(* Offers algorithms used to rank features. *)
	{attribute 'TcIecLibraryType'}
{attribute 'Namespace' := 'Tc3_Vision'}
TYPE ETcVnFeatureScoreTypeORB : (
	TCVN_FST_ORB_HARRIS:=0, 	(* Harris algorithm (produces more stable keypoints, but computation takes longer). *)
	TCVN_FST_ORB_FAST:=1	(* FAST algorithm (produces slightly less stable keypoints, but computation is faster). *)
) DINT;
END_TYPE

// Data Types/Enumerations/ETcVnFlipAxis

(* Defines the axis around which to flip (mirror) the image. *)
	{attribute 'TcIecLibraryType'}
{attribute 'Namespace' := 'Tc3_Vision'}
TYPE ETcVnFlipAxis : (
	TCVN_FA_XY:=-1, 	(* Flip the image around both axes *)
	TCVN_FA_X:=0, 	(* Flip the image around the X axis *)
	TCVN_FA_Y:=1	(* Flip the image around the Y axis *)
);
END_TYPE

// Data Types/Enumerations/ETcVnFilterDirection

(* Offers directions, in which to apply filter. *)
	{attribute 'TcIecLibraryType'}
{attribute 'Namespace' := 'Tc3_Vision'}
TYPE ETcVnFilterDirection : (
	TCVN_FD_X:=0, 	(* X-direction *)
	TCVN_FD_Y:=1	(* Y-direction *)
);
END_TYPE

// Data Types/Enumerations/ETcVnFontType

(* Offers font types. *)
	{attribute 'TcIecLibraryType'}
{attribute 'Namespace' := 'Tc3_Vision'}
TYPE ETcVnFontType : (
	TCVN_FT_HERSHEY_SIMPLEX:=0, 	(* Normal size sans-serif font. *)
	TCVN_FT_HERSHEY_PLAIN:=1, 	(* Small size sans-serif font. *)
	TCVN_FT_HERSHEY_DUPLEX:=2, 	(* More complex normal size sans-serif font. *)
	TCVN_FT_HERSHEY_COMPLEX:=3, 	(* Normal size serif font. *)
	TCVN_FT_HERSHEY_TRIPLEX:=4, 	(* More complex normal size serif font. *)
	TCVN_FT_HERSHEY_COMPLEX_SMALL:=5, 	(* Small size serif font. *)
	TCVN_FT_HERSHEY_SCRIPT_SIMPLEX:=6, 	(* Hand-writing style font. *)
	TCVN_FT_HERSHEY_SCRIPT_COMPLEX:=7, 	(* More complex hand-writing style font. *)
	TCVN_FT_HERSHEY_PLAIN_ITALIC:=17, 	(* Small size sans-serif font (italic). *)
	TCVN_FT_HERSHEY_COMPLEX_ITALIC:=19, 	(* Normal size serif font (italic). *)
	TCVN_FT_HERSHEY_TRIPLEX_ITALIC:=20, 	(* More complex normal size serif font (italic). *)
	TCVN_FT_HERSHEY_COMPLEX_SMALL_ITALIC:=21	(* Small size serif font (italic). *)
) DINT;
END_TYPE

// Data Types/Enumerations/ETcVnHoughMethod

(* Offers Hough methods. *)
	{attribute 'TcIecLibraryType'}
{attribute 'Namespace' := 'Tc3_Vision'}
TYPE ETcVnHoughMethod : (
	TCVN_HM_STANDARD:=0, 	(* Classical or standard Hough transform. Every line is represented by two floating-point numbers (f1, f2), where f1 is a distance between (0,0) origin and the line, and f2 is the angle between x-axis and the normal to the line. *)
	TCVN_HM_PROBABILISTIC:=1, 	(* Probabilistic Hough transform. More efficient for pictures containing long linear segments. Returns line segments rather than the whole line, while each segment is represented by start and end point. *)
	TCVN_HM_MULTI_SCALE:=2, 	(* Multi scale variant of classical Hough transform. *)
	TCVN_HM_GRADIENT:=3, 	(* Method designed to find circles. See paper: HK Yuen, John Princen, John Illingworth, and Josef Kittler. Comparative study of hough transform methods for circle finding. Image and Vision Computing, 8(1):71–77, 1990 *)
	TCVN_HM_GRADIENT_ALT:=4	(* Variation of the GRADIENT method. *)
) DINT;
END_TYPE

// Data Types/Enumerations/ETcVnInitializableFunction

(* Offers initializable functions. *)
	{attribute 'TcIecLibraryType'}
{attribute 'Namespace' := 'Tc3_Vision'}
TYPE ETcVnInitializableFunction : (
	TCVN_IF_OCR:=0, 	(* F_VN_OCR *)
		{attribute 'hide'}
TCVN_IF_CODEDETECTION:=1	(* F_VN_CODEDETECTION *)
) DINT;
END_TYPE

// Data Types/Enumerations/ETcVnInterpolationType

(* Offers interpolation types. *)
	{attribute 'TcIecLibraryType'}
{attribute 'Namespace' := 'Tc3_Vision'}
TYPE ETcVnInterpolationType : (
	TCVN_IT_NEAREST_NEIGHBOR:=0, 	(* Nearest neighbor interpolation *)
	TCVN_IT_BILINEAR:=1, 	(* Bilinear interpolation *)
	TCVN_IT_BICUBIC:=2, 	(* Bicubic interpolation *)
	TCVN_IT_AREA_BASED:=3, 	(* Area based interpolation *)
	TCVN_IT_LANCZOS4:=4	(* Lanczos4 interpolation *)
) DINT;
END_TYPE

// Data Types/Enumerations/ETcVnKnn

(* Offers kNN model types. *)
	{attribute 'TcIecLibraryType'}
{attribute 'Namespace' := 'Tc3_Vision'}
TYPE ETcVnKnn : (
	TCVN_KNN_CLASSIFIER:=1, 	(* Classifier *)
	TCVN_KNN_NOVELTY_DETECTOR:=2, 	(* Novelty detector *)
	TCVN_KNN_REGRESSOR:=4	(* Regressor *)
) UDINT;
END_TYPE

// Data Types/Enumerations/ETcVnLineType

(* Offers line types. *)
	{attribute 'TcIecLibraryType'}
{attribute 'Namespace' := 'Tc3_Vision'}
TYPE ETcVnLineType : (
	TCVN_LT_4_CONNECTED:=4, 	(* 4-connected (pixels are connected horizontally and vertically). *)
	TCVN_LT_8_CONNECTED:=8, 	(* 8-connected (pixels are connected horizontally, vertically and diagonally). *)
	TCVN_LT_ANTIALIASED:=16	(* Antialiased (drawn using Gaussian filtering, only implemented for 8-bit images). *)
) DINT;
END_TYPE

// Data Types/Enumerations/ETcVnMorphologicalOperator

(* Offers morphological operators. *)
	{attribute 'TcIecLibraryType'}
{attribute 'Namespace' := 'Tc3_Vision'}
TYPE ETcVnMorphologicalOperator : (
	TCVN_MO_EROSION:=16#0, 	(* Shrinks objects (regions of foreground (i.e. white) pixels), removing regions smaller than the structuring element completely. *)
	TCVN_MO_DILATION:=16#1, 	(* Expands objects and thereby closes small holes inside objects. *)
	TCVN_MO_OPENING:=16#2, 	(* Applies an erosion first, a dilation second. Objects smaller than the structuring element are removed while outer shapes remain largely the same. *)
	TCVN_MO_CLOSING:=16#3, 	(* Applies a dilation first, an erosion second. Holes inside objects that fit into the structuring element are closed completely while outer shapes remain largely the same. *)
	TCVN_MO_GRADIENT:=16#4, 	(* Difference between the dilation and the erosion of an image. *)
	TCVN_MO_WHITE_TOPHAT:=16#5, 	(* Difference between an input image and its opening. *)
	TCVN_MO_BLACK_TOPHAT:=16#6, 	(* Difference between an input image and its closing. *)
	TCVN_MO_OPENING_BY_RECONSTRUCTION:=16#40000002, 	(* Opening with subsequent reconstruction of objects that were not removed by the opening. *)
	TCVN_MO_CLOSING_BY_RECONSTRUCTION:=16#40000003, 	(* Closing with subsequent reconstruction of objects that were not removed by the closing. *)
	TCVN_MO_WHITE_TOPHAT_BY_RECONSTRUCTION:=16#40000005, 	(* White tophat with subsequent reconstruction of objects that were not removed by the white tophat. *)
	TCVN_MO_BLACK_TOPHAT_BY_RECONSTRUCTION:=16#40000006	(* Black tophat with subsequent reconstruction of objects that were not removed by the black tophat. *)
) DINT;
END_TYPE

// Data Types/Enumerations/ETcVnNbc

(* Offers normal Bayes classifier types. *)
	{attribute 'TcIecLibraryType'}
{attribute 'Namespace' := 'Tc3_Vision'}
TYPE ETcVnNbc : (
	TCVN_NBC_CLASSIFIER:=1, 	(* Classifier *)
	TCVN_NBC_NOVELTY_DETECTOR:=2	(* Novelty detector *)
) UDINT;
END_TYPE

// Data Types/Enumerations/ETcVnNormalizationType

(* Offers normalization types. *)
	{attribute 'TcIecLibraryType'}
{attribute 'Namespace' := 'Tc3_Vision'}
TYPE ETcVnNormalizationType : (
	TCVN_NT_INF:=1, 	(* Infinity norm *)
	TCVN_NT_L1:=2, 	(* L1 norm *)
	TCVN_NT_L2:=4, 	(* L2 (euclidean) norm *)
	TCVN_NT_L2SQR:=5, 	(* Squared L2 norm *)
	TCVN_NT_HAMMING:=6, 	(* Hamming distance (bitwise) *)
	TCVN_NT_HAMMING2:=7, 	(* Hamming distance (each 2 bits combined to one) *)
	TCVN_NT_RELATIVE_INF:=9, 	(* Infinity norm (when comparing 2 arrays, the norm of their difference is divided by the norm of the second array) *)
	TCVN_NT_RELATIVE_L1:=10, 	(* L1 norm (when comparing 2 arrays, the norm of their difference is divided by the norm of the second array) *)
	TCVN_NT_RELATIVE_L2:=12, 	(* L2 (euclidean) norm (when comparing 2 arrays, the norm of their difference is divided by the norm of the second array) *)
	TCVN_NT_RELATIVE_L2SQR:=13, 	(* Squared L2 norm (when comparing 2 arrays, the norm of their difference is divided by the norm of the second array) *)
	TCVN_NT_RELATIVE_HAMMING:=14, 	(* Hamming distance (bitwise; when comparing 2 arrays, the norm of their difference is divided by the norm of the second array) *)
	TCVN_NT_RELATIVE_HAMMING2:=15, 	(* Hamming distance (each 2 bits combined to one; when comparing 2 arrays, the norm of their difference is divided by the norm of the second array) *)
	TCVN_NT_MINMAX:=32	(* Normalize the values to a range given by a minimum and a maximum value. *)
) DINT;
END_TYPE

// Data Types/Enumerations/ETcVnFeatureScalingType

(* Offers feature scaling  types *)
	{attribute 'TcIecLibraryType'}
{attribute 'Namespace' := 'Tc3_Vision'}
TYPE ETcVnFeatureScalingType : (
	TCVN_FST1_MAXABS:=0, 	(* Use the max of the absolute values of the feature vector. The normlized values are in the range [-1 to 1] or [0 to 1] if all the original values are positive. *)
	TCVN_FST1_MINMAX:=1, 	(* Use the min and max values of the feature vector. The normlized values are in the range [0 to 1] *)
	TCVN_FST1_STANDARDIZATION:=2	(* Use the mean and the standard deviation of the feature vector. The normalized vector has a mean value equal to zero and standard deviation equal to one *)
) DINT;
END_TYPE

// Data Types/Enumerations/ETcVnOcrModelType

(* Offers different OCR model types *)
	{attribute 'TcIecLibraryType'}
{attribute 'Namespace' := 'Tc3_Vision'}
TYPE ETcVnOcrModelType : (
	TCVN_OMT_NUMBERS:=580542139465730, 	(* Classify numbers *)
	TCVN_OMT_NUMBERS_SC:=580542139465732, 	(* Classify numbers and special characters *)
	TCVN_OMT_UCLETTERS:=580542139465736, 	(* Classify uppercase letters *)
	TCVN_OMT_NUMBERS_SC_UCLETTERS:=580542139465744	(* Classify numbers, special characters and uppercase letters *)
) ULINT;
END_TYPE

// Data Types/Enumerations/ETcVnOcrOptions

(* Provides different options to indicate whether certain actions must be performed to achieve the intended result. *)
	{attribute 'TcIecLibraryType'}
{attribute 'Namespace' := 'Tc3_Vision'}
TYPE ETcVnOcrOptions : (
	TCVN_OO_NONE:=0, 	(* No options *)
	TCVN_OO_WITHBLANKS:=1	(* Indicates that if blanks were found, they should be included in the result. By default, all blanks are omitted from the result. *)
) UDINT;
END_TYPE

// Data Types/Enumerations/ETcVnOrientationMethod

(* Offers methods to calculate the orientation of a set of points. *)
	{attribute 'TcIecLibraryType'}
{attribute 'Namespace' := 'Tc3_Vision'}
TYPE ETcVnOrientationMethod : (
	TCVN_OM_PCA:=0, 	(* Apply the PCA on the points and calculate the mean point as the center point and the rotation angle of the main principal axis *)
	TCVN_OM_FITELLIPSE:=1, 	(* Fit an ellipse around the points and calculate the center point and the rotation angle of the main axis *)
	TCVN_OM_MOMENTS:=2, 	(* Calculate the moments of the points and estimate the center and the rotation angle *)
	TCVN_OM_ENCLOSINGRECT:=3	(* Calculate a minimum area rectangle enclosing the points and calculate the center point and the rotation angle of the rectangle *)
) DINT;
END_TYPE

// Data Types/Enumerations/ETcVnPaddingMode

(* Offers padding modes. *)
	{attribute 'TcIecLibraryType'}
{attribute 'Namespace' := 'Tc3_Vision'}
TYPE ETcVnPaddingMode : (
	TCVN_PM_NONE:=0, 	(* Resize the image to the desired size without extra processing *)
	TCVN_PM_CROP_CENTER:=1, 	(* Resize and crop the image *)
	TCVN_PM_LETTERBOX:=2	(* Resize the image to the desired size while preserving the aspect ratio of the original image *)
) DINT;
END_TYPE

// Data Types/Enumerations/ETcVnPixelConnectivity

(* Offers pixel connectivities. *)
	{attribute 'TcIecLibraryType'}
{attribute 'Namespace' := 'Tc3_Vision'}
TYPE ETcVnPixelConnectivity : (
	TCVN_PC_4:=4, 	(* 4-way *)
	TCVN_PC_8:=8	(* 8-way *)
) DINT;
END_TYPE

// Data Types/Enumerations/ETcVnPrototypeClusterer

(* Offers prototype clusterer model types. *)
	{attribute 'TcIecLibraryType'}
{attribute 'Namespace' := 'Tc3_Vision'}
TYPE ETcVnPrototypeClusterer : (
	TCVN_PC_NOVELTY_DETECTOR:=2, 	(* Novelty detector *)
	TCVN_PC_CLUSTERER:=8	(* Clusterer *)
) UDINT;
END_TYPE

// Data Types/Enumerations/ETcVnRectangleIntersection

(* Offers rectangle intersection types. *)
	{attribute 'TcIecLibraryType'}
{attribute 'Namespace' := 'Tc3_Vision'}
TYPE ETcVnRectangleIntersection : (
	TCVN_RI_NONE:=0, 	(* No intersection *)
	TCVN_RI_PARTIAL:=1, 	(* Partial intersection *)
	TCVN_RI_FULL:=2	(* Full intersection *)
) DINT;
END_TYPE

// Data Types/Enumerations/ETcVnRotationAngle

(* Offers rotation angles. *)
	{attribute 'TcIecLibraryType'}
{attribute 'Namespace' := 'Tc3_Vision'}
TYPE ETcVnRotationAngle : (
	TCVN_RA_90_DEG:=0, 	(* 90 degrees *)
	TCVN_RA_180_DEG:=1, 	(* 180 degrees *)
	TCVN_RA_270_DEG:=2	(* 270 degrees *)
) DINT;
END_TYPE

// Data Types/Enumerations/ETcVnRTrees

(* Offers RTrees model types. *)
	{attribute 'TcIecLibraryType'}
{attribute 'Namespace' := 'Tc3_Vision'}
TYPE ETcVnRTrees : (
	TCVN_RT_CLASSIFIER:=1, 	(* Classifier *)
	TCVN_RT_REGRESSOR:=4	(* Regressor *)
) UDINT;
END_TYPE

// Data Types/Enumerations/ETcVnSignedNormalization

(* Offers options for normalizing images with signed data types. *)
	{attribute 'TcIecLibraryType'}
{attribute 'Namespace' := 'Tc3_Vision'}
TYPE ETcVnSignedNormalization : (
	TCVN_SN_FIX_ZERO:=0, 	(* The value 0 is fixed, i.e. the normalized image might only reach either the minimum or maximum value. *)
	TCVN_SN_FULL_SCALE:=1	(* The image is normalized to the full value range, i.e. a prior value of 0 might be != 0 after normalization. *)
);
END_TYPE

// Data Types/Enumerations/ETcVnSolvePnPMethod

(* Offers SolvePnP methods. *)
	{attribute 'TcIecLibraryType'}
{attribute 'Namespace' := 'Tc3_Vision'}
TYPE ETcVnSolvePnPMethod : (
	TCVN_SPM_ITERATIVE:=0, 	(* Levenberg-Marquardt optimization. Requires at least 4 planar or 6 non-planar reference points. *)
	TCVN_SPM_EPNP:=1, 	(* Efficient perspective-n-point camera pose estimation. Requires at least 4 reference points. *)
	TCVN_SPM_P3P:=2, 	(* Complete solution classification for the perspective-three-point problem. Requires exactly 4 reference points to find a unique solution. *)
	TCVN_SPM_AP3P:=5, 	(* An efficient algebraic solution to the perspective-three-point problem. Requires exactly 4 reference points to find a unique solution. *)
	TCVN_SPM_IPPE:=6, 	(* Infinitesimal plane-based pose estimation. Requires at least 4 coplanar reference points. *)
	TCVN_SPM_IPPE_SQUARE:=7, 	(* IPPE specialization for squares. Requires exactly 4 reference points in the following order (hsl: half square length): (-hsl, hsl, 0), (hsl, hsl, 0), (hsl, -hsl, 0), (-hsl, -hsl, 0) *)
	TCVN_SPM_SQPNP:=8	(* A consistently fast and globally optimal solution to the perspective-n-point problem. Requires at least 4 reference points. *)
) DINT;
END_TYPE

// Data Types/Enumerations/ETcVnSta

(* Offers Simplified TopoART model types. *)
	{attribute 'TcIecLibraryType'}
{attribute 'Namespace' := 'Tc3_Vision'}
TYPE ETcVnSta : (
	TCVN_STA_CLASSIFIER:=1, 	(* Classifier *)
	TCVN_STA_NOVELTY_DETECTOR:=2, 	(* Novelty detector *)
	TCVN_STA_REGRESSOR:=4, 	(* Regressor *)
	TCVN_STA_CLUSTERER:=8	(* Clusterer *)
) UDINT;
END_TYPE

// Data Types/Enumerations/ETcVnStructuringElementShape

(* Offers shapes for a structuring element. *)
	{attribute 'TcIecLibraryType'}
{attribute 'Namespace' := 'Tc3_Vision'}
TYPE ETcVnStructuringElementShape : (
	TCVN_SES_RECTANGLE:=0, 	(* Rectangle *)
	TCVN_SES_CROSS:=1, 	(* Cross *)
	TCVN_SES_ELLIPSE:=2	(* Ellipse *)
) DINT;
END_TYPE

// Data Types/Enumerations/ETcVnSvm

(* Offers SVM model types. *)
	{attribute 'TcIecLibraryType'}
{attribute 'Namespace' := 'Tc3_Vision'}
TYPE ETcVnSvm : (
	TCVN_SVM_C_CLASSIFIER:=1, 	(* Classifier *)
	TCVN_SVM_NU_CLASSIFIER:=65537, 	(* Classifier *)
	TCVN_SVM_NOVELTY_DETECTOR:=2, 	(* Novelty detector *)
	TCVN_SVM_EPS_REGRESSOR:=4, 	(* Regressor *)
	TCVN_SVM_NU_REGRESSOR:=65540	(* Regressor *)
) UDINT;
END_TYPE

// Data Types/Enumerations/ETcVnSvmKernelType

(* Offers SVM kernel types. *)
	{attribute 'TcIecLibraryType'}
{attribute 'Namespace' := 'Tc3_Vision'}
TYPE ETcVnSvmKernelType : (
	TCVN_SKT_LINEAR:=0, 	(* Linear kernel (fast) *)
	TCVN_SKT_POLY:=1, 	(* Polynomial kernel *)
	TCVN_SKT_RBF:=2, 	(* Radial basis function (RBF) kernel (good default) *)
	TCVN_SKT_SIGMOID:=3, 	(* Sigmoid kernel *)
	TCVN_SKT_CHI2:=4, 	(* Chi-squared kernel *)
	TCVN_SKT_INTER:=5	(* Histogram intersection kernel *)
) DINT;
END_TYPE

// Data Types/Enumerations/ETcVnSvmSgdClassifierType

(* Offers different types of SVMSGD classifiers. *)
	{attribute 'TcIecLibraryType'}
{attribute 'Namespace' := 'Tc3_Vision'}
TYPE ETcVnSvmSgdClassifierType : (
	TCVN_SSCT_SGD:=0, 	(* Stochastic Gradient Descent *)
	TCVN_SSCT_ASGD:=1	(* Average Stochastic Gradient Descent *)
) DINT;
END_TYPE

// Data Types/Enumerations/ETcVnSvmSgdClassifierMarginType

(* Offers different margin types for SVMSGD classifiers. *)
	{attribute 'TcIecLibraryType'}
{attribute 'Namespace' := 'Tc3_Vision'}
TYPE ETcVnSvmSgdClassifierMarginType : (
	TCVN_SSCMT_SOFT_MARGIN:=0, 	(* Soft margin allowing outliers. (beneficial for classes that cannot be separated linearly) *)
	TCVN_SSCMT_HARD_MARGIN:=1	(* Hard margin. (best-suited for linearly separable classes) *)
) DINT;
END_TYPE

// Data Types/Enumerations/ETcVnTemplateMatchMethod

(* Offers methods for template matching. *)
	{attribute 'TcIecLibraryType'}
{attribute 'Namespace' := 'Tc3_Vision'}
TYPE ETcVnTemplateMatchMethod : (
	TCVN_TMM_SQDIFF:=0, 	(* Squared difference (supports template mask) *)
	TCVN_TMM_SQDIFF_NORMED:=1, 	(* Normalized squared difference *)
	TCVN_TMM_CCORR:=2, 	(* Cross-correlation *)
	TCVN_TMM_CCORR_NORMED:=3, 	(* Normalized cross-correlation (supports template mask) *)
	TCVN_TMM_CCOEFF:=4, 	(* Correlation coefficient *)
	TCVN_TMM_CCOEFF_NORMED:=5	(* Normalized correlation coefficient *)
) DINT;
END_TYPE

// Data Types/Enumerations/ETcVnThresholdType

(* Offers threshold types. *)
	{attribute 'TcIecLibraryType'}
{attribute 'Namespace' := 'Tc3_Vision'}
TYPE ETcVnThresholdType : (
	TCVN_TT_BINARY:=0, 	(* Binary threshold *)
	TCVN_TT_BINARY_INV:=1, 	(* Inverted binary threshold *)
	TCVN_TT_TRUNC:=2, 	(* Truncated threshold (pixels > thresh are set to thresh, others keep their value) *)
	TCVN_TT_TOZERO:=3, 	(* To zero threshold (pixels < thresh are set to zero, others keep their value) *)
	TCVN_TT_TOZERO_INV:=4, 	(* Inverted to zero threshold (pixels > thresh are set to zero, others keep their value) *)
	TCVN_TT_OTSU_BINARY:=8, 	(* Binary threshold with the threshold value selected according to the Otsu algorithm *)
	TCVN_TT_OTSU_BINARY_INV:=9, 	(* Inverted binary threshold with the threshold value selected according to the Otsu algorithm *)
	TCVN_TT_OTSU_TRUNC:=10, 	(* Truncated threshold with the threshold value selected according to the Otsu algorithm *)
	TCVN_TT_OTSU_TOZERO:=11, 	(* To zero threshold with the threshold value selected according to the Otsu algorithm *)
	TCVN_TT_OTSU_TOZERO_INV:=12, 	(* Inverted to zero threshold with the threshold value selected according to the Otsu algorithm *)
	TCVN_TT_TRIANGLE_BINARY:=16, 	(* Binary threshold with the threshold value selected according to the Triangle algorithm *)
	TCVN_TT_TRIANGLE_BINARY_INV:=17, 	(* Inverted binary threshold with the threshold value selected according to the Triangle algorithm *)
	TCVN_TT_TRIANGLE_TRUNC:=18, 	(* Truncated threshold with the threshold value selected according to the Triangle algorithm *)
	TCVN_TT_TRIANGLE_TOZERO:=19, 	(* To zero threshold with the threshold value selected according to the Triangle algorithm *)
	TCVN_TT_TRIANGLE_TOZERO_INV:=20	(* Inverted to zero threshold with the threshold value selected according to the Triangle algorithm *)
) DINT;
END_TYPE

// Data Types/Enumerations/ETcVnTimestamp

(* Offers image acquisition timestamps. *)
	{attribute 'TcIecLibraryType'}
{attribute 'Namespace' := 'Tc3_Vision'}
TYPE ETcVnTimestamp : (
	TCVN_TS_IMAGE_COMPLETED:=1	(* Timestamp when the image was completed, i.e. all packets were received by the GigEVision driver. *)
) ULINT;
END_TYPE

// Data Types/Enumerations/ETcVnVectorCompareMethod

(* Offers methods for vector comparison. *)
	{attribute 'TcIecLibraryType'}
{attribute 'Namespace' := 'Tc3_Vision'}
TYPE ETcVnVectorCompareMethod : (
	TCVN_VCM_EUCLIDEAN:=0, 	(* Euclidean *)
	TCVN_VCM_ELEMENTWISE:=1	(* Elementwise *)
) DINT;
END_TYPE

// Data Types/Enumerations/ETcVnKeypointDetectionTypeAGAST

(* Offers different neighborhood types for AGAST method (For details see paper: E. Mair et al.: Adaptive and Generic Corner Detection Based on the Accelerated Segment Test, 2010). *)
	{attribute 'TcIecLibraryType'}
{attribute 'Namespace' := 'Tc3_Vision'}
TYPE ETcVnKeypointDetectionTypeAGAST : (
	TCVN_KDT_AGAST_5_8:=0, 	(* 5 of 8 *)
	TCVN_KDT_AGAST_7_12d:=1, 	(* 7 of 12 diamond *)
	TCVN_KDT_AGAST_7_12s:=2, 	(* 7 of 12 square *)
	TCVN_KDT_AGAST_9_16:=3	(* 9 of 16 *)
) DINT;
END_TYPE

// Data Types/Enumerations/ETcVnKeypointDetectionTypeFAST

(* Offers different neighborhood types for FAST method (For details see paper: E. Rosten: Machine Learning for High-speed Corner Detection, 2006). *)
	{attribute 'TcIecLibraryType'}
{attribute 'Namespace' := 'Tc3_Vision'}
TYPE ETcVnKeypointDetectionTypeFAST : (
	TCVN_KDT_FAST_5_8:=0, 	(* 5 of 8 *)
	TCVN_KDT_FAST_7_12:=1, 	(* 7 of 12 *)
	TCVN_KDT_FAST_9_16:=2	(* 9 of 16 *)
) DINT;
END_TYPE

// Data Types/Enumerations/ETcVnWorldCoordinateSystem

(* Offers world coordinate system orientations. *)
	{attribute 'TcIecLibraryType'}
{attribute 'Namespace' := 'Tc3_Vision'}
TYPE ETcVnWorldCoordinateSystem : (
	TCVN_WCS_X_RIGHT_Y_DOWN:=0, 	(* X axis points right, Y axis down (same orientation as image coordinate system) *)
	TCVN_WCS_X_DOWN_Y_RIGHT:=1, 	(* X axis points down, Y axis right *)
	TCVN_WCS_X_LEFT_Y_DOWN:=2, 	(* X axis points left, Y axis down *)
	TCVN_WCS_X_UP_Y_RIGHT:=3, 	(* X axis points up, Y axis right *)
	TCVN_WCS_X_RIGHT_Y_UP:=4, 	(* X axis points right, Y axis up *)
	TCVN_WCS_X_DOWN_Y_LEFT:=5, 	(* X axis points down, Y axis left *)
	TCVN_WCS_X_LEFT_Y_UP:=6, 	(* X axis points left, Y axis up *)
	TCVN_WCS_X_UP_Y_LEFT:=7	(* X axis points up, Y axis left *)
) DINT;
END_TYPE

// Data Types/Structs/TcVnCodeGrades1D

(* Describes code quality grades for 1D barcodes according to ISO / IEC 15416:2016. The grades range from 0 (very bad) to 4 (very good) and are averaged over several scan lines. *)
	{attribute 'TcIecLibraryType'}
{attribute 'Namespace' := 'Tc3_Vision'}
TYPE TcVnCodeGrades1D : 
	STRUCT
		(* Decode grade *)
		fDecode : REAL;
		(* Symbol contrast grade *)
		fSymbolContrast : REAL;
		(* Minimum reflectance grade *)
		fMinReflectance : REAL;
		(* Minimum edge contrast grade *)
		fMinEdgeContrast : REAL;
		(* Modulation grade *)
		fModulation : REAL;
		(* Defects grade *)
		fDefects : REAL;
		(* Decodability grade *)
		fDecodability : REAL;
		(* Overall code grade, i.e. the minimum achieved individual grade averaged over all scan lines. If different scan lines lead to different decoded data, the overall grade is 0. *)
		fOverall : REAL;
	END_STRUCT
END_TYPE

// Data Types/Structs/TcVnCodeGradesDM

(* Describes code quality grades for Data Matrix codes according to ISO / IEC 15415:2011. The grades range from 0 (very bad) to 4 (very good). *)
	{attribute 'TcIecLibraryType'}
{attribute 'Namespace' := 'Tc3_Vision'}
TYPE TcVnCodeGradesDM : 
	STRUCT
		(* Decode grade *)
		nDecode : USINT;
		(* Symbol contrast grade *)
		nSymbolContrast : USINT;
		(* Modulation grade *)
		nModulation : USINT;
		(* Reflectance margin grade *)
		nReflectanceMargin : USINT;
		(* Fixed pattern damage grade *)
		nFixedPatternDamage : USINT;
		(* Axial nonuniformity grade *)
		nAxialNonuniformity : USINT;
		(* Grid nonuniformity grade *)
		nGridNonuniformity : USINT;
		(* Unused error correction grade *)
		nUnusedErrorCorrection : USINT;
		(* Overall code grade, i.e. the minimum achieved individual grade *)
		nOverall : USINT;
	END_STRUCT
END_TYPE

// Data Types/Structs/TcVnCodeGradesQR

(* Describes code quality grades for QR codes according to ISO / IEC 15415:2011. The grades range from 0 (very bad) to 4 (very good). *)
	{attribute 'TcIecLibraryType'}
{attribute 'Namespace' := 'Tc3_Vision'}
TYPE TcVnCodeGradesQR : 
	STRUCT
		(* Decode grade *)
		nDecode : USINT;
		(* Symbol contrast grade *)
		nSymbolContrast : USINT;
		(* Modulation grade *)
		nModulation : USINT;
		(* Reflectance margin grade *)
		nReflectanceMargin : USINT;
		(* Fixed pattern damage grade *)
		nFixedPatternDamage : USINT;
		(* Axial nonuniformity grade *)
		nAxialNonuniformity : USINT;
		(* Grid nonuniformity grade *)
		nGridNonuniformity : USINT;
		(* Unused error correction grade *)
		nUnusedErrorCorrection : USINT;
		(* Format information grade *)
		nFormatInfo : USINT;
		(* Version information grade *)
		nVersionInfo : USINT;
		(* Overall code grade, i.e. the minimum achieved individual grade *)
		nOverall : USINT;
	END_STRUCT
END_TYPE

// Data Types/Structs/TcVnParamsAGAST

(* Offers parameters for AGAST method. *)
	{attribute 'TcIecLibraryType'}
{attribute 'Namespace' := 'Tc3_Vision'}
TYPE TcVnParamsAGAST : 
	STRUCT
		(* Threshold for the intensity difference between the center pixel and its surrounding circle *)
		nThreshold : DINT := 10;
		(* If true, non-maximum suppression is applied. *)
		bNonMaxSuppression : BOOL := TRUE;
		 {attribute 'hide'}
		_reserved1 : ARRAY [1..3] OF USINT;
		(* Neighborhood type *)
		 {attribute 'GUID' := 'FA6F5C56-A2E3-4BCD-8022-41680719FF8A'}
		 {attribute 'Namespace' := 'Tc3_Vision'}
		eType : ETcVnKeypointDetectionTypeAGAST := TCVN_KDT_AGAST_9_16;
	END_STRUCT
END_TYPE

// Data Types/Structs/TcVnParamsAKAZE

(* Offers parameters for AKAZE method. *)
	{attribute 'TcIecLibraryType'}
{attribute 'Namespace' := 'Tc3_Vision'}
TYPE TcVnParamsAKAZE : 
	STRUCT
		(* Type of the descriptor *)
		 {attribute 'GUID' := 'EFB57555-E4E6-46A8-8672-7CE1494D9FAA'}
		 {attribute 'Namespace' := 'Tc3_Vision'}
		eDescrType : ETcVnFeatureDescriptorTypeAKAZE := TCVN_FDT_AKAZE_MLDB;
		(* Size of the descriptor in bits (only for MLDB; 0 = full size) *)
		nDescrSize : UDINT := 0;
		(* Number of descriptor channels (currently only 3 supported for MLDB) *)
		nDescrChannels : UDINT := 3;
		(* Detector response threshold *)
		fThreshold : REAL := 0.001;
		(* Maximum octave evolution *)
		nOctaves : UDINT := 2;
		(* Number of sublevels per scale level *)
		nOctaveLayers : UDINT := 1;
		(* Diffusivity type *)
		 {attribute 'GUID' := '808733BC-B2E0-4793-A0CE-2F414F4C0F1D'}
		 {attribute 'Namespace' := 'Tc3_Vision'}
		eDiffusivity : ETcVnDiffusivityTypeKAZE := TCVN_DT1_KAZE_PM_G2;
	END_STRUCT
END_TYPE

// Data Types/Structs/TcVnParamsBlobDetection

(* Offers parameters for blob detection *)
	{attribute 'TcIecLibraryType'}
{attribute 'Namespace' := 'Tc3_Vision'}
TYPE TcVnParamsBlobDetection : 
	STRUCT
		(* Enable filtering by area (fMinArea <= area <= fMaxArea); strongly recommended to activate for filtering noise with fMinArea. *)
		bFilterByArea : BOOL := TRUE;
		(* Enable filtering by circularity (fMinCircularity <= circularity(4pi * area / perimeter^2) <= fMaxCircularity). *)
		bFilterByCircularity : BOOL := FALSE;
		(* Enable filtering by convexity (fMinConvexity <= convexity(area / hullArea) <= fMaxConvexity). *)
		bFilterByConvexity : BOOL := FALSE;
		(* Enable filtering by eccentricity (fMinEccentricity <= eccentricity <= fMaxEccentricity). *)
		bFilterByEccentricity : BOOL := FALSE;
		(* Enable filtering by inertia ratio (fMinInertiaRatio <= inertia ratio <= fMaxInertiaRatio). *)
		bFilterByInertiaRatio : BOOL := FALSE;
		 {attribute 'hide'}
		_reserved1 : ARRAY [1..3] OF USINT;
		(* Min estimated blob area in pixel *)
		fMinArea : REAL := 10;
		(* Max estimated blob area in pixel *)
		fMaxArea : REAL := 100000000;
		(* Min circularity (1.0: ideal circle, < 1: less circular, 0: not circular at all) *)
		fMinCircularity : REAL := 0;
		(* Max circularity (1.0: ideal circle, < 1: less circular, 0: not circular at all) *)
		fMaxCircularity : REAL := 1;
		(* Min convexity (1.0: blob fully convex, < 1: less convex) *)
		fMinConvexity : REAL := 0;
		(* Max convexity (1.0: blob fully convex, < 1: less convex) *)
		fMaxConvexity : REAL := 1;
		(* Min eccentricity (0.0: circular, 1.0: linear) *)
		fMinEccentricity : REAL := 0;
		(* Max eccentricity (0.0: circular, 1.0: linear) *)
		fMaxEccentricity : REAL := 1;
		(* Min inertia ratio (1.0: equal width and height, 0.0: linear) *)
		fMinInertiaRatio : REAL := 0;
		(* Max inertia ratio (1.0: equal width and height, 0.0: linear) *)
		fMaxInertiaRatio : REAL := 1;
		(* Threshold type for internally applied threshold method (OTSU_XXX only supported for USINT images). *)
		 {attribute 'GUID' := 'C40D9A7B-C720-49F8-A5B9-1663BB6925B6'}
		 {attribute 'Namespace' := 'Tc3_Vision'}
		eThresholdType : ETcVnThresholdType := TCVN_TT_BINARY;
		(* Threshold to start with (if fThresholdStep > 0, otherwise this is the only threshold used). *)
		fMinThreshold : REAL := 30;
		(* Threshold to end with (if fThresholdStep > 0, otherwise this value is not used). *)
		fMaxThreshold : REAL := 225;
		(* Sets to 0 if only 1 threshold should be used (much faster than multiple thresholds and combining the results). *)
		fThresholdStep : REAL := 0;
		(* Minimum distance between the center points of two different blobs (only used if fThresholdStep > 0; if distance < fMinBlobDistance, the blobs are treated as the same). *)
		fMinBlobDistance : REAL := 5;
		(* Minimum number of threshold steps, for which the same contour has to be detected (only used if fThresholdStep > 0; same means center point distance < fMinBlobDistance). *)
		nMinRepeatability : UDINT := 2;
		(* Selects, which of the multi-threshold blob contours should be returned. *)
		 {attribute 'GUID' := '6B3EA399-FB72-4A3D-A347-965F9D388EB6'}
		 {attribute 'Namespace' := 'Tc3_Vision'}
		eBlobCombination : ETcVnBlobCombination := TCVN_BC_MEDIAN_THRESHOLD;
	END_STRUCT
END_TYPE

// Data Types/Structs/TcVnParamsBRISK

(* Offers parameters for BRISK method. *)
	{attribute 'TcIecLibraryType'}
{attribute 'Namespace' := 'Tc3_Vision'}
TYPE TcVnParamsBRISK : 
	STRUCT
		(* Detection threshold *)
		nThreshold : DINT := 30;
		(* Detection octaves (0 for single scale) *)
		nOctaves : UDINT := 3;
		(* Scale factor for the neighborhood pattern *)
		fPatternScale : REAL := 1;
	END_STRUCT
END_TYPE

// Data Types/Structs/TcVnParamsFAST

(* Offers parameters for FAST method. *)
	{attribute 'TcIecLibraryType'}
{attribute 'Namespace' := 'Tc3_Vision'}
TYPE TcVnParamsFAST : 
	STRUCT
		(* Threshold for the intensity difference between the center pixel and its surrounding circle *)
		nThreshold : DINT := 10;
		(* If true, non-maximum suppression is applied. *)
		bNonMaxSuppression : BOOL := TRUE;
		 {attribute 'hide'}
		_reserved1 : ARRAY [1..3] OF USINT;
		(* Neighborhood type *)
		 {attribute 'GUID' := 'FBD32F44-42B6-42E8-8896-D6A6C0F64387'}
		 {attribute 'Namespace' := 'Tc3_Vision'}
		eType : ETcVnKeypointDetectionTypeFAST := TCVN_KDT_FAST_9_16;
	END_STRUCT
END_TYPE

// Data Types/Structs/TcVnParamsGFTT

(* Offers parameters for GFTT method. *)
	{attribute 'TcIecLibraryType'}
{attribute 'Namespace' := 'Tc3_Vision'}
TYPE TcVnParamsGFTT : 
	STRUCT
		(* Maximum number of corners to return (strongest ones) *)
		nMaxCorners : UDINT := 1000;
		 {attribute 'hide'}
		_reserved1 : UDINT;
		(* Minimum accepted corner quality, relative to the strongest one *)
		fQualityLevel : LREAL := 0.01;
		(* Minimum euclidean distance between returned keypoints *)
		fMinDistance : LREAL := 1;
		(* Neighborhood block size *)
		nBlockSize : UDINT := 3;
		(* If true, a Harris detector is used instead of the default method. *)
		bUseHarrisDetector : BOOL := FALSE;
		 {attribute 'hide'}
		_reserved2 : ARRAY [1..3] OF USINT;
		(* Free parameter of the Harris detector *)
		fHarrisK : LREAL := 0.04;
	END_STRUCT
END_TYPE

// Data Types/Structs/TcVnParamsKAZE

(* Offers parameters for KAZE method *)
	{attribute 'TcIecLibraryType'}
{attribute 'Namespace' := 'Tc3_Vision'}
TYPE TcVnParamsKAZE : 
	STRUCT
		(* If true, the descriptor size is extended from the default 64 byte to 128 byte. *)
		bExtended : BOOL := FALSE;
		(* If true, upright (rotation dependent) descriptors are computed. *)
		bUpright : BOOL := FALSE;
		 {attribute 'hide'}
		_reserved1 : UINT;
		(* Detector response threshold *)
		fThreshold : REAL := 0.001;
		(* Maximum octave evolution of the image *)
		nOctaves : UDINT := 4;
		(* Number of sublevels per scale level *)
		nOctaveLayers : UDINT := 2;
		(* Diffusivity type *)
		 {attribute 'GUID' := '808733BC-B2E0-4793-A0CE-2F414F4C0F1D'}
		 {attribute 'Namespace' := 'Tc3_Vision'}
		eDiffusivity : ETcVnDiffusivityTypeKAZE := TCVN_DT1_KAZE_PM_G2;
	END_STRUCT
END_TYPE

// Data Types/Structs/TcVnParamsMSER

(* Offers parameters for MSER method *)
	{attribute 'TcIecLibraryType'}
{attribute 'Namespace' := 'Tc3_Vision'}
TYPE TcVnParamsMSER : 
	STRUCT
		(* Delta for size comparison *)
		nDelta : DINT := 5;
		(* Minimum blob size *)
		nMinArea : UDINT := 60;
		(* Maximum blob size *)
		nMaxArea : UDINT := 14400;
		 {attribute 'hide'}
		_reserved1 : UDINT;
		(* Maximum blob size variation *)
		fMaxVariation : LREAL := 0.25;
		(* Minimum MSER diversity *)
		fMinDiversity : LREAL := 0.2;
		(* Maximum evolution steps (only used for color images) *)
		nMaxEvolution : UDINT := 200;
		 {attribute 'hide'}
		_reserved2 : UDINT;
		(* Area threshold to cause re-initialization (only used for color images) *)
		fAreaThreshold : LREAL := 1.01;
		(* Minimum margin (only used for color images) *)
		fMinMargin : LREAL := 0.003;
		(* Aperture size for edge bluring (only used for color images) *)
		nEdgeBlurSize : UDINT := 5;
		 {attribute 'hide'}
		_reserved3 : UDINT;
	END_STRUCT
END_TYPE

// Data Types/Structs/TcVnParamsORB

(* Offers parameters for ORB method. *)
	{attribute 'TcIecLibraryType'}
{attribute 'Namespace' := 'Tc3_Vision'}
TYPE TcVnParamsORB : 
	STRUCT
		(* Maximum number of returned keypoints *)
		nMaxPoints : UDINT := 500;
		(* Pyramid decimation ratio (must be greater than 1, should be smaller than 2) *)
		fPyramidScale : REAL := 1.2;
		(* Number of pyramid levels *)
		nPyramidLevels : UDINT := 8;
		(* Size of the border, where no features are detected (should match nPatchSize) *)
		nEdgeThreshold : UDINT := 31;
		(* First pyramid level (currently, only 0 is supported) *)
		nFirstLevel : UDINT := 0;
		(* Number of points to produce each BRIEF descriptor element (2, 3, 4) *)
		nBriefPoints : UDINT := 2;
		(* Score type (HARRIS is more stable but slightly slower than FAST) *)
		 {attribute 'GUID' := '688ACEF5-9A4A-4447-9B39-CBC4558C02DB'}
		 {attribute 'Namespace' := 'Tc3_Vision'}
		eScoreType : ETcVnFeatureScoreTypeORB := TCVN_FST_ORB_HARRIS;
		(* Patch size of the BRIEF descriptor *)
		nPatchSize : UDINT := 31;
		(* Threshold for the FAST keypoint detection *)
		nFastThreshold : DINT := 20;
	END_STRUCT
END_TYPE

// Data Types/Structs/TcVnParamsSB

(* Offers parameters for SB method (a simple blob detector with multiple thresholds). *)
	{attribute 'TcIecLibraryType'}
{attribute 'Namespace' := 'Tc3_Vision'}
TYPE TcVnParamsSB : 
	STRUCT
		(* Enable filtering by area (fMinArea <= area < fMaxArea). *)
		bFilterByArea : BOOL := TRUE;
		(* Enable filtering by circularity (fMinCircularity <= circularity(4pi * area / perimeter^2) < fMaxCircularity). *)
		bFilterByCircularity : BOOL := FALSE;
		(* Enable filtering by color (thresholdedColor(0 or 255) = nBlobColor). *)
		bFilterByColor : BOOL := FALSE;
		(* Enable filtering by convexity (fMinConvexity <= convexity(area / hullArea) < fMaxConvexity). *)
		bFilterByConvexity : BOOL := FALSE;
		(* Enable filtering by inertia ratio (fMinInertiaRatio <= inertia ratio < fMaxInertiaRatio). *)
		bFilterByInertia : BOOL := FALSE;
		 {attribute 'hide'}
		_reserved1 : ARRAY [1..3] OF USINT;
		(* Min estimated blob area in pixel *)
		fMinArea : REAL := 25;
		(* Max estimated blob area in pixel *)
		fMaxArea : REAL := 15000;
		(* Min circularity (1.0: ideal circle, < 1: less circular, 0: not circular at all) *)
		fMinCircularity : REAL := 0;
		(* Max circularity (1.0: ideal circle, < 1: less circular, 0: not circular at all) *)
		fMaxCircularity : REAL := 1;
		(* 0 or 255 *)
		nBlobColor : USINT := 255;
		 {attribute 'hide'}
		_reserved2 : ARRAY [1..3] OF USINT;
		(* Min convexity (1.0: blob fully convex, < 1: less convex) *)
		fMinConvexity : REAL := 0;
		(* Max convexity (1.0: blob fully convex, < 1: less convex) *)
		fMaxConvexity : REAL := 1;
		(* Min inertia ratio (0.0 .. 1.0) *)
		fMinInertiaRatio : REAL := 0;
		(* Max inertia ratio (0.0 .. 1.0) *)
		fMaxInertiaRatio : REAL := 1;
		(* Min distance between different blobs *)
		fMinBlobDist : REAL := 5;
		(* Min number of same detected blobs (dist < fMinBlobDist) in different thresholds *)
		nMinRepeatability : UDINT := 2;
		(* Min threshold (start) *)
		fMinThreshold : REAL := 30;
		(* Max threshold (stop) *)
		fMaxThreshold : REAL := 225;
		(* Threshold step between min and max threshold *)
		fThresholdStep : REAL := 10;
	END_STRUCT
END_TYPE

// Version/Global_Version
{attribute 'TcGenerated'}
// This function has been automatically generated from the project information.
VAR_GLOBAL CONSTANT
	{attribute 'const_non_replaced'}
	{attribute 'linkalways'}
	stLibVersion_Tc3_Vision : ST_LibVersion := (iMajor := 5, iMinor := 5, iBuild := 10, iRevision := 0, sVersion := '5.5.10.0');
	{attribute 'const_non_replaced'}
	{attribute 'linkalways'}
	sLibraryId_Tc3_Vision : String := 'Beckhoff Automation GmbH|Tc3_Vision|5.5.10.0';
END_VAR

// Global Variables/Global_Variables

	VAR_GLOBAL
		VISION_ADS_TIMEOUT	:	TIME := TIME#5s;	(* Default ADS timeout. *)
	END_VAR

// Global Variables/TC3_VISION_IID_LIST

	VAR_GLOBAL
		IID_ITcVnColorModel	:	IID := (Data1 := 16#AFF801F3, Data2 := 16#60D0, Data3 := 16#43FA, Data4 := [16#98, 16#0F, 16#57, 16#2A, 16#62, 16#05, 16#B5, 16#AF]);	(* Interface ID for interface ITcVnColorModel *)
	END_VAR

// Function Blocks/Image Acquisition/FB_VN_GevCameraControl

	{attribute 'c++_compatible'}
	{attribute 'external_name' := 'FB_VN_GevCameraControl_GUID_E0C38C9A_95D7_4F88_D282_FD5E0D0B8646'}
	{attribute 'TcIecLibraryType'}
	{attribute 'no_explicit_call' :='do not call this POU directly'}
	(* This FB provides the basic functionality to control a GigE Vision camera and access its calibration data. *)
	FUNCTION_BLOCK FB_VN_GevCameraControl
	VAR
		(* Internal reference to the corresponding TcVnGevImageProvider TcCOM module ID, which needs to be set via TC init symbol. *)
		{attribute 'TcInitSymbol'}
		{attribute 'TcCategoryOID' := 'TcVnGevImageProvider'}
		 {attribute 'GUID' := '18071995-0000-0000-0000-00000000000F'}
		oidITcVnGevImageProvider : OTCID;
		 {attribute 'hide'}
		_reserved1 : UINT_0_32;
		(* Internal stuff *)
		{attribute 'hide'}
		 {attribute 'GUID' := '18071995-0000-0000-0000-000000000018'}
		pInternal : PVOID;
	END_VAR


	(* Delete all images contained in the TcVnGevImageProvider TcCOM module receive queue and reset the corresponding omitted images counter. *)
	METHOD ClearImageQueue : HRESULT
END_METHOD


	(* Close the control channel to the camera. *)
	METHOD CloseCamera : HRESULT
END_METHOD


	(* Internal method *)
	{attribute 'hide'}
	METHOD FB_exit : BOOL
	VAR_INPUT
		(*  if TRUE, the exit method is called for exiting an instance that is copied afterwards (online change). *)
		bInCopyCode : BOOL;
	END_VAR
END_METHOD


	(* Internal method *)
	{attribute 'hide'}
	METHOD FB_init : BOOL
	VAR_INPUT
		(*  if TRUE, the retain variables are initialized (warm start / cold start) *)
		bInitRetains : BOOL;
		(*  if TRUE, the instance afterwards gets moved into the copy code (online change) *)
		bInCopyCode : BOOL;
	END_VAR
END_METHOD


	(* Gets the reference calibration pattern points from the TcVnGevImageProvider TcCOM module (Can be set from the calibration assistant) *)
	METHOD GetCalibPatternRef : HRESULT
	VAR_INPUT
		(* Returns the reference calibration pattern points (ContainerType_Vector_TcVnPoint3_REAL) *)
 {attribute 'GUID' := 'BC72B333-E095-465B-9693-7979773CA3B8'}
				ipCalibPatternRef : REFERENCE TO ITcVnContainer;
	END_VAR
END_METHOD


	(* Gets the camera matrix from the TcVnGevImageProvider TcCOM module (requires intrinsic calibration parameters, e.g. set by the calibration assistant) *)
	METHOD GetCameraMatrix : HRESULT
	VAR_IN_OUT
		(* Returns the camera matrix *)
 {attribute 'GUID' := '91A420A3-4727-4481-B3BB-170528E5BC7C'}
		 {attribute 'Namespace' := 'VN'}
				aCameraMatrix : TcVnMatrix3x3_LREAL;
	END_VAR
END_METHOD


	(* Gets the current available image (first in receive queue). *)
	METHOD GetCurrentImage : HRESULT
	VAR_INPUT
		(* Returns the image *)
 {attribute 'GUID' := '70D42C6D-6F4E-4719-8B29-2883D5D59B1C'}
				ipImage : REFERENCE TO ITcVnImage;
	END_VAR
END_METHOD


	(* Gets the current available image (first in receive queue) with undistortion applied. Incompatible with pixel formats that contain an encoding, e.g. a Bayer pattern. Requires intrinsic calibration parameters in the TcVnGevImageProvider TcCOM module, e.g. set by the calibration assistant. *)
	METHOD GetCurrentImageUndistorted : HRESULT
	VAR_INPUT
		(* Returns the undistorted image *)
 {attribute 'GUID' := '70D42C6D-6F4E-4719-8B29-2883D5D59B1C'}
				ipImage : REFERENCE TO ITcVnImage;
	END_VAR
END_METHOD


	(* Gets the current available image (first in receive queue) and its corresponding GVSP info. *)
	METHOD GetCurrentImageWithGvspInfo : HRESULT
	VAR_INPUT
		(* Returns the image *)
 {attribute 'GUID' := '70D42C6D-6F4E-4719-8B29-2883D5D59B1C'}
				ipImage : REFERENCE TO ITcVnImage;
	END_VAR
	VAR_IN_OUT
		(* Returns the GVSP info *)
 {attribute 'GUID' := '63FC7E33-91CD-44CD-9015-0BD1DC25722C'}
				stGvspInfo : GVSP_IMAGE_INFO;
	END_VAR
END_METHOD


	(* Gets the current available image (first in receive queue) with its corresponding GVSP info and undistortion applied. Incompatible with pixel formats that contain an encoding, e.g. a Bayer pattern. Requires intrinsic calibration parameters in the TcVnGevImageProvider TcCOM module, e.g. set by the calibration assistant. *)
	METHOD GetCurrentImageWithGvspInfoUndistorted : HRESULT
	VAR_INPUT
		(* Returns the undistorted image *)
 {attribute 'GUID' := '70D42C6D-6F4E-4719-8B29-2883D5D59B1C'}
				ipImage : REFERENCE TO ITcVnImage;
	END_VAR
	VAR_IN_OUT
		(* Returns the GVSP info *)
 {attribute 'GUID' := '63FC7E33-91CD-44CD-9015-0BD1DC25722C'}
				stGvspInfo : GVSP_IMAGE_INFO;
	END_VAR
END_METHOD


	(* Gets the current available image (first in receive queue) and corresponding timestamps. *)
	METHOD GetCurrentImageWithTimestamps : HRESULT
	VAR_INPUT
		(* Returns the image *)
 {attribute 'GUID' := '70D42C6D-6F4E-4719-8B29-2883D5D59B1C'}
				ipImage : REFERENCE TO ITcVnImage;
		(* Select timestamps to return (ETcVnTimestamp) *)
		nTimestamps : ULINT;
		(* Returns the requested timestamps (make sure to provide an array of sufficient size). *)
		pTimestamps : POINTER TO LINT;
	END_VAR
	VAR_OUTPUT
		(* Returns the GVSP info *)
 {attribute 'GUID' := '63FC7E33-91CD-44CD-9015-0BD1DC25722C'}
				stGvspInfo : GVSP_IMAGE_INFO;
	END_VAR
END_METHOD


	(* Gets the distortion coefficients from the TcVnGevImageProvider TcCOM module (requires intrinsic calibration parameters, e.g. set by the calibration assistant) *)
	METHOD GetDistortionCoefficients : HRESULT
	VAR_IN_OUT
		(* Returns the distortion coefficients [k1, k2, p1, p2, k3, k4, k5, k6] *)
 {attribute 'GUID' := 'DD112102-C23A-4B37-A43A-A96400B57010'}
		 {attribute 'Namespace' := 'VN'}
				aDistortionCoefficients : TcVnArray8_LREAL;
	END_VAR
END_METHOD


	(* Gets the last received image from the queue. *)
	METHOD GetLastImageFromQueue : HRESULT
	VAR_INPUT
		(* Returns the image *)
 {attribute 'GUID' := '70D42C6D-6F4E-4719-8B29-2883D5D59B1C'}
				ipImage : REFERENCE TO ITcVnImage;
	END_VAR
END_METHOD


	(* Gets the number of omitted images since the last call of ClearImageQueue(). If the image receive queue in the TcVnGevImageProvider TcCOM module is full and a new image arrives, the first one in the queue will be deleted and the omitted counter is increased. *)
	METHOD GetOmittedImagesNum : HRESULT
	VAR_IN_OUT
		(* Returns the number of omitted images *)
		nOmitted : ULINT;
	END_VAR
END_METHOD


	(* Gets the rotation matrix from the TcVnGevImageProvider TcCOM module (requires extrinsic calibration parameters, e.g. set by the calibration assistant) *)
	METHOD GetRotationMatrix : HRESULT
	VAR_IN_OUT
		(* Returns the rotation matrix *)
 {attribute 'GUID' := '91A420A3-4727-4481-B3BB-170528E5BC7C'}
		 {attribute 'Namespace' := 'VN'}
				aRotationMatrix : TcVnMatrix3x3_LREAL;
	END_VAR
END_METHOD


	(* Gets the current state of the internal camera control state machine. *)
	METHOD GetState : ETcVnCameraState
END_METHOD


	(* Gets the translation vector from the TcVnGevImageProvider TcCOM module (requires extrinsic calibration parameters, e.g. set by the calibration assistant) *)
	METHOD GetTranslationVector : HRESULT
	VAR_IN_OUT
		(* Returns the translation vector *)
 {attribute 'GUID' := 'B9A67DEB-A7D1-4F25-95A3-4A82FA5C1E28'}
		 {attribute 'Namespace' := 'VN'}
				aTranslationVector : TcVnVector3_LREAL;
	END_VAR
END_METHOD


	(* Initialize the camera to the intended state (includes sending the 'InitCameraCommands' defined in the GevImageAcquisition TcCOM module to the camera). *)
	METHOD InitializeCamera : HRESULT
END_METHOD


	(* Open a control channel to the camera. *)
	METHOD OpenCamera : HRESULT
END_METHOD


	(* Reset the camera controller to initial state (might require multiple calls depending on current state, until S_OK is returned) *)
	METHOD Reset : HRESULT
END_METHOD


	(* Reset the camera features to initial state (sends the 'InitCameraCommands' defined in the GevImageAcquisition TcCOM module to the camera). *)
	METHOD ResetCameraFeatures : HRESULT
END_METHOD


	(* Sets the camera matrix to the TcVnGevImageProvider TcCOM module *)
	METHOD SetCameraMatrix : HRESULT
	VAR_IN_OUT
		(* The camera matrix to be copied to the TcCOM module *)
 {attribute 'GUID' := '91A420A3-4727-4481-B3BB-170528E5BC7C'}
		 {attribute 'Namespace' := 'VN'}
				aCameraMatrix : TcVnMatrix3x3_LREAL;
	END_VAR
END_METHOD


	(* Sets the distortion coefficients to the TcVnGevImageProvider TcCOM module *)
	METHOD SetDistortionCoefficients : HRESULT
	VAR_IN_OUT
		(* The distortion coefficients to be copied to the TcCOM module *)
 {attribute 'GUID' := 'DD112102-C23A-4B37-A43A-A96400B57010'}
		 {attribute 'Namespace' := 'VN'}
				aDistortionCoefficients : TcVnArray8_LREAL;
	END_VAR
END_METHOD


	(* Sets the rotation matrix to the TcVnGevImageProvider TcCOM module *)
	METHOD SetRotationMatrix : HRESULT
	VAR_IN_OUT
		(* The rotation matrix to be copied to the TcCOM module *)
 {attribute 'GUID' := '91A420A3-4727-4481-B3BB-170528E5BC7C'}
		 {attribute 'Namespace' := 'VN'}
				aRotationMatrix : TcVnMatrix3x3_LREAL;
	END_VAR
END_METHOD


	(* Sets the translation vector to the TcVnGevImageProvider TcCOM module *)
	METHOD SetTranslationVector : HRESULT
	VAR_IN_OUT
		(* The translation vector to be copied to the TcCOM module *)
 {attribute 'GUID' := 'B9A67DEB-A7D1-4F25-95A3-4A82FA5C1E28'}
		 {attribute 'Namespace' := 'VN'}
				aTranslationVector : TcVnVector3_LREAL;
	END_VAR
END_METHOD


	(* Send the 'StartAcquisitionCommands' defined in the TcVnGevImageProvider TcCOM module to the camera. *)
	METHOD StartAcquisition : HRESULT
END_METHOD


	(* Send the 'StopAcquisitionCommands' defined in the TcVnGevImageProvider TcCOM module to the camera. *)
	METHOD StopAcquisition : HRESULT
END_METHOD


	(* Send the 'SoftwareTriggerCommands' defined in the TcVnGevImageProvider TcCOM module to the camera. *)
	METHOD TriggerImage : HRESULT
END_METHOD

END_FUNCTION_BLOCK

// Function Blocks/Image Acquisition/FB_VN_FileSourceControl

	{attribute 'c++_compatible'}
	{attribute 'external_name' := 'FB_VN_FileSourceControl_GUID_BF1EF806_AD3C_426D_E484_B59DB5FAA980'}
	{attribute 'TcIecLibraryType'}
	{attribute 'no_explicit_call' :='do not call this POU directly'}
	(* This FB provides access to the images send by a File Source instance. *)
	FUNCTION_BLOCK FB_VN_FileSourceControl
	VAR
		(* Internal reference to the corresponding TcVnFileImageProvider TcCOM module ID, which needs to be set via TC init symbol. *)
		{attribute 'TcInitSymbol'}
		{attribute 'TcCategoryOID' := 'TcVnFileImageProvider'}
		 {attribute 'GUID' := '18071995-0000-0000-0000-00000000000F'}
		oidITcVnFileImageProvider : OTCID;
		 {attribute 'hide'}
		_reserved1 : UINT_0_32;
		(* Internal reference to private data. *)
		{attribute 'hide'}
		 {attribute 'GUID' := '18071995-0000-0000-0000-000000000018'}
		pPriv : PVOID;
	END_VAR


	(* Internal method *)
	{attribute 'hide'}
	METHOD FB_exit : BOOL
	VAR_INPUT
		(* If TRUE, the exit method is called for exiting an instance that is copied afterwards (online change). *)
		bInCopyCode : BOOL;
	END_VAR
END_METHOD


	(* Internal method *)
	{attribute 'hide'}
	METHOD FB_init : BOOL
	VAR_INPUT
		(* If TRUE, the retain variables are initialized (warm start / cold start) *)
		bInitRetains : BOOL;
		(* If TRUE, the exit method is called for exiting an instance that is copied afterwards (online change). *)
		bInCopyCode : BOOL;
	END_VAR
END_METHOD


	(* Gets the current available image (if any). *)
	METHOD GetCurrentImage : HRESULT
	VAR_INPUT
		(* Returns the image *)
 {attribute 'GUID' := '70D42C6D-6F4E-4719-8B29-2883D5D59B1C'}
				ipImage : REFERENCE TO ITcVnImage;
	END_VAR
END_METHOD


	(* Gets the current available image (if any) and the corresponding file name. *)
	METHOD GetCurrentImageAndFileName : HRESULT
	VAR_INPUT
		(* Returns the image *)
 {attribute 'GUID' := '70D42C6D-6F4E-4719-8B29-2883D5D59B1C'}
				ipImage : REFERENCE TO ITcVnImage;
	END_VAR
	VAR_IN_OUT CONSTANT
		(* Returns the file name *)
 {attribute 'GUID' := '18071995-0000-0000-0000-00000000001A'}
				sFileName : STRING;
	END_VAR
	VAR_INPUT
		(* Define the maximum allowed length for the file name *)
		nMaxLen : UINT;
	END_VAR
END_METHOD


	(* Activates the File Source. If not in trigger mode, it will start sending images. *)
	METHOD StartAcquisition : HRESULT
END_METHOD


	(* Deactivates the File Source. It will stop sending images. *)
	METHOD StopAcquisition : HRESULT
END_METHOD


	(* Reset the controller to initial state (might require multiple calls depending on current state, until S_OK is returned) *)
	METHOD Reset : HRESULT
END_METHOD


	(* Gets the current state of the internal camera control state machine. *)
	METHOD GetState : ETcVnCameraState
END_METHOD


	(* If in trigger mode, this function triggers the next image in the list. *)
	METHOD TriggerImage : HRESULT
END_METHOD


	(* If in trigger mode, this function triggers a specific image in the list. *)
	METHOD TriggerImageExp : HRESULT
	VAR_INPUT
		(* Amount of images to skip, relative to current *)
		nSkipImages : DINT;
	END_VAR
END_METHOD


	(* If in trigger mode, this function triggers a specific image in the list by name. *)
	METHOD TriggerImageByName : HRESULT
	VAR_IN_OUT CONSTANT
		(* Name of the image to trigger *)
 {attribute 'GUID' := '18071995-0000-0000-0000-00000000001A'}
				sImageName : STRING;
	END_VAR
END_METHOD

END_FUNCTION_BLOCK

// Function Blocks/Image Acquisition/FB_VN_SimpleCameraControl

	{attribute 'c++_compatible'}
	{attribute 'external_name' := 'FB_VN_SimpleCameraControl_GUID_3530661D_FCB1_48FD_F78A_F761ECBA890C'}
	{attribute 'TcIecLibraryType'}
	{attribute 'no_explicit_call' :='do not call this POU directly'}
	(* This FB provides the basic functionality to control a camera or a FileSource. *)
	FUNCTION_BLOCK FB_VN_SimpleCameraControl
	VAR
		(* Internal reference to the corresponding TcVnImageProvider TcCOM module ID, which needs to be set via TC init symbol. *)
		{attribute 'TcInitSymbol'}
		{attribute 'TcCategoryOID' := 'TcVnImageProvider'}
		 {attribute 'GUID' := '18071995-0000-0000-0000-00000000000F'}
		oidITcVnImageProvider : OTCID;
		 {attribute 'hide'}
		_reserved1 : UINT_0_32;
		(* Internal stuff *)
		{attribute 'hide'}
		 {attribute 'GUID' := '18071995-0000-0000-0000-000000000018'}
		pInternal : PVOID;
	END_VAR


	(* Internal method *)
	{attribute 'hide'}
	METHOD FB_exit : BOOL
	VAR_INPUT
		(*  if TRUE, the exit method is called for exiting an instance that is copied afterwards (online change). *)
		bInCopyCode : BOOL;
	END_VAR
END_METHOD


	(* Internal method *)
	{attribute 'hide'}
	METHOD FB_init : BOOL
	VAR_INPUT
		(*  if TRUE, the retain variables are initialized (warm start / cold start) *)
		bInitRetains : BOOL;
		(*  if TRUE, the instance afterwards gets moved into the copy code (online change) *)
		bInCopyCode : BOOL;
	END_VAR
END_METHOD


	(* Get the current available image (if any). *)
	METHOD GetCurrentImage : HRESULT
	VAR_INPUT
		(* Returns the image *)
 {attribute 'GUID' := '70D42C6D-6F4E-4719-8B29-2883D5D59B1C'}
				ipImage : REFERENCE TO ITcVnImage;
	END_VAR
END_METHOD


	(* Get the current state of the internal camera control state machine. *)
	METHOD GetState : ETcVnCameraState
END_METHOD


	(* Reset the camera to initial state (might require multiple calls depending on current state, until S_OK is returned) *)
	METHOD Reset : HRESULT
END_METHOD


	(* Start the image acquisition. *)
	METHOD StartAcquisition : HRESULT
END_METHOD


	(* Stop the image acquisition. *)
	METHOD StopAcquisition : HRESULT
END_METHOD


	(* Trigger the next image. *)
	METHOD TriggerImage : HRESULT
END_METHOD

END_FUNCTION_BLOCK

// Function Blocks/File Access/FB_VN_InitializeFunction

	{attribute 'c++_compatible'}
	{attribute 'external_name' := 'FB_VN_InitializeFunction_GUID_C13A97AB_8F2F_4225_FF15_35BCADA0C9FC'}
	{attribute 'TcIecLibraryType'}
	(* This FB initializes selected functions. Before, it needs to initialize itself, i.e. call the FB until the output bInitialized is true before using it for function initialization. *)
	FUNCTION_BLOCK FB_VN_InitializeFunction
	VAR_INPUT
		(* Selects the function to initialize *)
		 {attribute 'GUID' := 'E6ED44CE-C5A2-4A6C-A74A-99081CD9253B'}
		 {attribute 'Namespace' := 'Tc3_Vision'}
		eFunction : ETcVnInitializableFunction;
	END_VAR
	VAR
		 {attribute 'hide'}
		_reserved1 : UINT_0_32;
	END_VAR
	VAR_INPUT
		(* Selects initialization options for the function *)
		nOptions : ULINT := 0;
		(* Function initialization is triggered by a rising edge at this input. *)
		bStart : BOOL;
	END_VAR
	VAR
		 {attribute 'hide'}
		_reserved2 : ARRAY [1..3] OF USINT;
	END_VAR
	VAR_INPUT
		(* Indicates the time before the function is cancelled. *)
		nTimeout : TIME := VISION_ADS_TIMEOUT;
	END_VAR
	VAR_OUTPUT
		(* This output remains TRUE until the function block has executed a command, but at the longest for the duration supplied to the 'nTimeout' input. While bBusy = TRUE, no new command will be accepted at the inputs. *)
		bBusy : BOOL;
		(* This output is switched to TRUE as soon as an error occurs during the execution of a command. The command-specific error code is contained in ‘nErrorId’. If the function block has a timeout error, 'bError' is TRUE and 'nErrorId' is 1861 (hexadecimal 0x745). Is reset to FALSE by the execution of a command at the inputs. *)
		bError : BOOL;
	END_VAR
	VAR
		 {attribute 'hide'}
		_reserved3 : UINT;
	END_VAR
	VAR_OUTPUT
		(* Contains the ADS error code or the command-specific error code of the last executed command. Is reset to 0 by the execution of a command at the inputs. *)
		nErrorId : UDINT;
	END_VAR
	VAR
		(* Internal parameter *)
		{attribute 'hide'}
		nAdsInvStamp : UINT;
		(* Internal parameter *)
		{attribute 'hide'}
		nAdsInvCnt : BYTE;
		(* Internal parameter *)
		{attribute 'hide'}
		ePendingRequest : BYTE;
		(* Internal parameter *)
		{attribute 'hide'}
		nTimeElapsed : TIME;
		(* Internal parameter *)
		{attribute 'hide'}
		bLastRead : BOOL;
		 {attribute 'hide'}
		_reserved4 : UINT_24_56;
		(* Internal parameter *)
		{attribute 'hide'}
		 {attribute 'GUID' := '18071995-0000-0000-0000-000000000018'}
		pBuffer : PVOID;
		(* Internal parameter *)
		{attribute 'hide'}
		 {attribute 'GUID' := 'E6ED44CE-C5A2-4A6C-A74A-99081CD9253B'}
		 {attribute 'Namespace' := 'Tc3_Vision'}
		ePendingFunction : ETcVnInitializableFunction;
		 {attribute 'hide'}
		_reserved5 : UDINT;
		(* Internal parameter *)
		{attribute 'hide'}
		nPendingOptions : ULINT;
		(* Internal parameter *)
		{attribute 'hide'}
		 {attribute 'GUID' := '18071995-0000-0000-0000-000000000018'}
		pFilePathPending : PVOID;
		(* Internal parameter *)
		{attribute 'hide'}
		nFilePathCounter : DINT;
		 {attribute 'hide'}
		_reserved6 : UINT_0_32;
	END_VAR


	(* Internal method *)
	{attribute 'hide'}
	METHOD FB_exit : BOOL
	VAR_INPUT
		(*  if TRUE, the exit method is called for exiting an instance that is copied afterwards (online change). *)
		bInCopyCode : BOOL;
	END_VAR
END_METHOD


	(* Internal method *)
	{attribute 'hide'}
	METHOD FB_init : BOOL
	VAR_INPUT
		(*  if TRUE, the retain variables are initialized (warm start / cold start) *)
		bInitRetains : BOOL;
		(*  if TRUE, the instance afterwards gets moved into the copy code (online change) *)
		bInCopyCode : BOOL;
	END_VAR
END_METHOD

END_FUNCTION_BLOCK

// Function Blocks/File Access/FB_VN_ReadCalibrationPattern

	{attribute 'c++_compatible'}
	{attribute 'external_name' := 'FB_VN_ReadCalibrationPattern_GUID_0334E03E_2BBE_407D_E2A1_068B13B2E811'}
	{attribute 'TcIecLibraryType'}
	(* This FB reads calibration pattern reference points from an xml file on the targte pc. *)
	FUNCTION_BLOCK FB_VN_ReadCalibrationPattern
	VAR_IN_OUT CONSTANT
		(* Full path of the file or relative path to the default directory on the target pc *)
		 {attribute 'GUID' := '18071995-0000-0000-0000-00000000001A'}
		sFilePath : STRING;
	END_VAR
	VAR_INPUT
		(* Returns a container with the pattern points (ContainerType_Vector_TcVnPoint3_REAL) *)
		 {attribute 'GUID' := 'BC72B333-E095-465B-9693-7979773CA3B8'}
		ipDestContainer : REFERENCE TO ITcVnContainer;
		(* Reading the file is triggered by a rising edge at this input. *)
		bRead : BOOL;
	END_VAR
	VAR
		 {attribute 'hide'}
		_reserved1 : ARRAY [1..3] OF USINT;
	END_VAR
	VAR_INPUT
		(* Indicates the time before the function is cancelled. *)
		nTimeout : TIME := VISION_ADS_TIMEOUT;
	END_VAR
	VAR_OUTPUT
		(* This output remains TRUE until the function block has executed a command, but at the longest for the duration supplied to the 'nTimeout' input. While bBusy = TRUE, no new command will be accepted at the inputs. *)
		bBusy : BOOL;
		(* This output is switched to TRUE as soon as an error occurs during the execution of a command. The command-specific error code is contained in ‘nErrorId’. If the function block has a timeout error, 'bError' is TRUE and 'nErrorId' is 1861 (hexadecimal 0x745). Is reset to FALSE by the execution of a command at the inputs. *)
		bError : BOOL;
	END_VAR
	VAR
		 {attribute 'hide'}
		_reserved2 : UINT;
	END_VAR
	VAR_OUTPUT
		(* Contains the ADS error code or the command-specific error code of the last executed command. Is reset to 0 by the execution of a command at the inputs. *)
		nErrorId : UDINT;
	END_VAR
	VAR
		(* Internal parameter *)
		{attribute 'hide'}
		nAdsInvStamp : UINT;
		(* Internal parameter *)
		{attribute 'hide'}
		nAdsInvCnt : BYTE;
		(* Internal parameter *)
		{attribute 'hide'}
		ePendingRequest : BYTE;
		(* Internal parameter *)
		{attribute 'hide'}
		nTimeElapsed : TIME;
		(* Internal parameter *)
		{attribute 'hide'}
		bLastRead : BOOL;
		 {attribute 'hide'}
		_reserved3 : UINT_24_56;
		(* Internal parameter *)
		{attribute 'hide'}
		 {attribute 'GUID' := '18071995-0000-0000-0000-000000000018'}
		pBuffer : PVOID;
		(* Internal parameter *)
		{attribute 'hide'}
		 {attribute 'GUID' := '18071995-0000-0000-0000-000000000018'}
		pFilePathPending : PVOID;
	END_VAR


	(* Internal method *)
	{attribute 'hide'}
	METHOD FB_exit : BOOL
	VAR_INPUT
		(*  if TRUE, the exit method is called for exiting an instance that is copied afterwards (online change). *)
		bInCopyCode : BOOL;
	END_VAR
END_METHOD


	(* Internal method *)
	{attribute 'hide'}
	METHOD FB_init : BOOL
	VAR_INPUT
		(*  if TRUE, the retain variables are initialized (warm start / cold start) *)
		bInitRetains : BOOL;
		(*  if TRUE, the instance afterwards gets moved into the copy code (online change) *)
		bInCopyCode : BOOL;
	END_VAR
END_METHOD

END_FUNCTION_BLOCK

// Function Blocks/File Access/FB_VN_ReadCalibrationResult

	{attribute 'c++_compatible'}
	{attribute 'external_name' := 'FB_VN_ReadCalibrationResult_GUID_EE7898B1_588B_4444_D687_3E4CD4FF96B9'}
	{attribute 'TcIecLibraryType'}
	(* This FB reads calibration results from a json file on the targte pc. *)
	FUNCTION_BLOCK FB_VN_ReadCalibrationResult
	VAR_IN_OUT CONSTANT
		(* Full path of the file or relative path to the default directory on the target pc *)
		 {attribute 'GUID' := '18071995-0000-0000-0000-00000000001A'}
		sFilePath : STRING;
	END_VAR
	VAR_INPUT
		(* Returns the camera matrix *)
		 {attribute 'GUID' := '91A420A3-4727-4481-B3BB-170528E5BC7C'}
		 {attribute 'Namespace' := 'VN'}
		aCameraMatrix : REFERENCE TO TcVnMatrix3x3_LREAL;
		(* Returns the distortion coefficients *)
		 {attribute 'GUID' := 'DD112102-C23A-4B37-A43A-A96400B57010'}
		 {attribute 'Namespace' := 'VN'}
		aDistortionCoefficients : REFERENCE TO TcVnArray8_LREAL;
		(* Returns the rotation matrix *)
		 {attribute 'GUID' := '91A420A3-4727-4481-B3BB-170528E5BC7C'}
		 {attribute 'Namespace' := 'VN'}
		aRotationMatrix : REFERENCE TO TcVnMatrix3x3_LREAL;
		(* Returns the translation vector *)
		 {attribute 'GUID' := 'B9A67DEB-A7D1-4F25-95A3-4A82FA5C1E28'}
		 {attribute 'Namespace' := 'VN'}
		aTranslationVector : REFERENCE TO TcVnVector3_LREAL;
		(* Reading the file is triggered by a rising edge at this input. *)
		bRead : BOOL;
	END_VAR
	VAR
		 {attribute 'hide'}
		_reserved1 : ARRAY [1..3] OF USINT;
	END_VAR
	VAR_INPUT
		(* Indicates the time before the function is cancelled. *)
		nTimeout : TIME := VISION_ADS_TIMEOUT;
	END_VAR
	VAR_OUTPUT
		(* This output remains TRUE until the function block has executed a command, but at the longest for the duration supplied to the 'nTimeout' input. While bBusy = TRUE, no new command will be accepted at the inputs. *)
		bBusy : BOOL;
		(* This output is switched to TRUE as soon as an error occurs during the execution of a command. The command-specific error code is contained in ‘nErrorId’. If the function block has a timeout error, 'bError' is TRUE and 'nErrorId' is 1861 (hexadecimal 0x745). Is reset to FALSE by the execution of a command at the inputs. *)
		bError : BOOL;
	END_VAR
	VAR
		 {attribute 'hide'}
		_reserved2 : UINT;
	END_VAR
	VAR_OUTPUT
		(* Contains the ADS error code or the command-specific error code of the last executed command. Is reset to 0 by the execution of a command at the inputs. *)
		nErrorId : UDINT;
	END_VAR
	VAR
		(* Internal parameter *)
		{attribute 'hide'}
		nAdsInvStamp : UINT;
		(* Internal parameter *)
		{attribute 'hide'}
		nAdsInvCnt : BYTE;
		(* Internal parameter *)
		{attribute 'hide'}
		ePendingRequest : BYTE;
		(* Internal parameter *)
		{attribute 'hide'}
		nTimeElapsed : TIME;
		(* Internal parameter *)
		{attribute 'hide'}
		bLastRead : BOOL;
		 {attribute 'hide'}
		_reserved3 : UINT_24_56;
		(* Internal parameter *)
		{attribute 'hide'}
		 {attribute 'GUID' := '18071995-0000-0000-0000-000000000018'}
		pBuffer : PVOID;
		(* Internal parameter *)
		{attribute 'hide'}
		 {attribute 'GUID' := '18071995-0000-0000-0000-000000000018'}
		pFilePathPending : PVOID;
	END_VAR


	(* Internal method *)
	{attribute 'hide'}
	METHOD FB_exit : BOOL
	VAR_INPUT
		(*  if TRUE, the exit method is called for exiting an instance that is copied afterwards (online change). *)
		bInCopyCode : BOOL;
	END_VAR
END_METHOD


	(* Internal method *)
	{attribute 'hide'}
	METHOD FB_init : BOOL
	VAR_INPUT
		(*  if TRUE, the retain variables are initialized (warm start / cold start) *)
		bInitRetains : BOOL;
		(*  if TRUE, the instance afterwards gets moved into the copy code (online change) *)
		bInCopyCode : BOOL;
	END_VAR
END_METHOD

END_FUNCTION_BLOCK

// Function Blocks/File Access/FB_VN_ReadContainer

	{attribute 'c++_compatible'}
	{attribute 'external_name' := 'FB_VN_ReadContainer_GUID_F9E4F2F1_F63B_40DB_DBB4_38C4670651B2'}
	{attribute 'TcIecLibraryType'}
	(* This FB reads a container from an xml file on the target pc. *)
	FUNCTION_BLOCK FB_VN_ReadContainer
	VAR_IN_OUT CONSTANT
		(* Full path of the file or relative path to the default directory on the target pc *)
		 {attribute 'GUID' := '18071995-0000-0000-0000-00000000001A'}
		sFilePath : STRING;
	END_VAR
	VAR_INPUT
		(* Returns a container with the loaded content *)
		 {attribute 'GUID' := 'BC72B333-E095-465B-9693-7979773CA3B8'}
		ipDestContainer : REFERENCE TO ITcVnContainer;
		(* The type id of the container to return. If this parameter is not set, a suitable container type will be determined automatically (except for csv files). *)
		 {attribute 'GUID' := '18071995-0000-0000-0000-000000000021'}
		nDestTypeGuid : GUID;
		(* Reading the file is triggered by a rising edge at this input. *)
		bRead : BOOL;
	END_VAR
	VAR
		 {attribute 'hide'}
		_reserved1 : ARRAY [1..3] OF USINT;
	END_VAR
	VAR_INPUT
		(* Indicates the time before the function is cancelled. *)
		nTimeout : TIME := VISION_ADS_TIMEOUT;
	END_VAR
	VAR_OUTPUT
		(* This output remains TRUE until the function block has executed a command, but at the longest for the duration supplied to the 'nTimeout' input. While bBusy = TRUE, no new command will be accepted at the inputs. *)
		bBusy : BOOL;
		(* This output is switched to TRUE as soon as an error occurs during the execution of a command. The command-specific error code is contained in ‘nErrorId’. If the function block has a timeout error, 'bError' is TRUE and 'nErrorId' is 1861 (hexadecimal 0x745). Is reset to FALSE by the execution of a command at the inputs. *)
		bError : BOOL;
	END_VAR
	VAR
		 {attribute 'hide'}
		_reserved2 : UINT;
	END_VAR
	VAR_OUTPUT
		(* Contains the ADS error code or the command-specific error code of the last executed command. Is reset to 0 by the execution of a command at the inputs. *)
		nErrorId : UDINT;
	END_VAR
	VAR
		(* Internal parameter *)
		{attribute 'hide'}
		nAdsInvStamp : UINT;
		(* Internal parameter *)
		{attribute 'hide'}
		nAdsInvCnt : BYTE;
		(* Internal parameter *)
		{attribute 'hide'}
		ePendingRequest : BYTE;
		(* Internal parameter *)
		{attribute 'hide'}
		nTimeElapsed : TIME;
		(* Internal parameter *)
		{attribute 'hide'}
		bLastRead : BOOL;
		 {attribute 'hide'}
		_reserved3 : UINT_24_56;
		(* Internal parameter *)
		{attribute 'hide'}
		 {attribute 'GUID' := '18071995-0000-0000-0000-000000000018'}
		pReadBuffer : PVOID;
		(* Internal parameter *)
		{attribute 'hide'}
		 {attribute 'GUID' := '18071995-0000-0000-0000-000000000018'}
		pWriteBuffer : PVOID;
		(* Internal parameter *)
		{attribute 'hide'}
		nWriteSize : UDINT;
		 {attribute 'hide'}
		_reserved4 : UINT_0_32;
	END_VAR


	(* Internal method *)
	{attribute 'hide'}
	METHOD FB_exit : BOOL
	VAR_INPUT
		(*  if TRUE, the exit method is called for exiting an instance that is copied afterwards (online change). *)
		bInCopyCode : BOOL;
	END_VAR
END_METHOD


	(* Internal method *)
	{attribute 'hide'}
	METHOD FB_init : BOOL
	VAR_INPUT
		(*  if TRUE, the retain variables are initialized (warm start / cold start) *)
		bInitRetains : BOOL;
		(*  if TRUE, the instance afterwards gets moved into the copy code (online change) *)
		bInCopyCode : BOOL;
	END_VAR
END_METHOD

END_FUNCTION_BLOCK

// Function Blocks/File Access/FB_VN_ReadImage

	{attribute 'c++_compatible'}
	{attribute 'external_name' := 'FB_VN_ReadImage_GUID_6CB69850_8BD3_4036_C664_818012EDC289'}
	{attribute 'TcIecLibraryType'}
	(* This FB reads an image from a file on the target pc. *)
	FUNCTION_BLOCK FB_VN_ReadImage
	VAR_IN_OUT CONSTANT
		(* Full path of the file or relative path to the default image directory on the target pc *)
		 {attribute 'GUID' := '18071995-0000-0000-0000-00000000001A'}
		sFilePath : STRING;
	END_VAR
	VAR_INPUT
		(* Returns an image with the loaded content *)
		 {attribute 'GUID' := '70D42C6D-6F4E-4719-8B29-2883D5D59B1C'}
		ipDestImage : REFERENCE TO ITcVnImage;
		(* Reading the file is triggered by a rising edge at this input. *)
		bRead : BOOL;
	END_VAR
	VAR
		 {attribute 'hide'}
		_reserved1 : ARRAY [1..3] OF USINT;
	END_VAR
	VAR_INPUT
		(* Indicates the time before the function is cancelled. *)
		nTimeout : TIME := VISION_ADS_TIMEOUT;
	END_VAR
	VAR_OUTPUT
		(* This output remains TRUE until the function block has executed a command, but at the longest for the duration supplied to the 'nTimeout' input. While bBusy = TRUE, no new command will be accepted at the inputs. *)
		bBusy : BOOL;
		(* This output is switched to TRUE as soon as an error occurs during the execution of a command. The command-specific error code is contained in ‘nErrorId’. If the function block has a timeout error, 'bError' is TRUE and 'nErrorId' is 1861 (hexadecimal 0x745). Is reset to FALSE by the execution of a command at the inputs. *)
		bError : BOOL;
	END_VAR
	VAR
		 {attribute 'hide'}
		_reserved2 : UINT;
	END_VAR
	VAR_OUTPUT
		(* Contains the ADS error code or the command-specific error code of the last executed command. Is reset to 0 by the execution of a command at the inputs. *)
		nErrorId : UDINT;
	END_VAR
	VAR
		(* Internal parameter *)
		{attribute 'hide'}
		nAdsInvStamp : UINT;
		(* Internal parameter *)
		{attribute 'hide'}
		nAdsInvCnt : BYTE;
		(* Internal parameter *)
		{attribute 'hide'}
		ePendingRequest : BYTE;
		(* Internal parameter *)
		{attribute 'hide'}
		nTimeElapsed : TIME;
		(* Internal parameter *)
		{attribute 'hide'}
		bLastRead : BOOL;
		 {attribute 'hide'}
		_reserved3 : UINT_24_56;
		(* Internal parameter *)
		{attribute 'hide'}
		 {attribute 'GUID' := '18071995-0000-0000-0000-000000000018'}
		pBuffer : PVOID;
		(* Internal parameter *)
		{attribute 'hide'}
		 {attribute 'GUID' := '18071995-0000-0000-0000-000000000018'}
		pFilePathPending : PVOID;
	END_VAR


	(* Internal method *)
	{attribute 'hide'}
	METHOD FB_exit : BOOL
	VAR_INPUT
		(*  if TRUE, the exit method is called for exiting an instance that is copied afterwards (online change). *)
		bInCopyCode : BOOL;
	END_VAR
END_METHOD


	(* Internal method *)
	{attribute 'hide'}
	METHOD FB_init : BOOL
	VAR_INPUT
		(*  if TRUE, the retain variables are initialized (warm start / cold start) *)
		bInitRetains : BOOL;
		(*  if TRUE, the instance afterwards gets moved into the copy code (online change) *)
		bInCopyCode : BOOL;
	END_VAR
END_METHOD

END_FUNCTION_BLOCK

// Function Blocks/File Access/FB_VN_ReadMlModel

	{attribute 'c++_compatible'}
	{attribute 'external_name' := 'FB_VN_ReadMlModel_GUID_B06841BB_6605_43B0_DA37_0B1728BAAC87'}
	{attribute 'TcIecLibraryType'}
	(* This FB reads a machine learning model from a file on the target pc. *)
	FUNCTION_BLOCK FB_VN_ReadMlModel
	VAR_IN_OUT CONSTANT
		(* Full path of the file or relative path to the default directory on the target pc *)
		 {attribute 'GUID' := '18071995-0000-0000-0000-00000000001A'}
		sFilePath : STRING;
	END_VAR
	VAR_INPUT
		(* Returns the loaded machine learning model *)
		 {attribute 'GUID' := 'AC23D64B-CDFA-4D43-AE8B-364A856EB3E2'}
		ipDestMlModel : REFERENCE TO ITcVnMlModel;
		(* Reading the file is triggered by a rising edge at this input. *)
		bRead : BOOL;
	END_VAR
	VAR
		 {attribute 'hide'}
		_reserved1 : ARRAY [1..3] OF USINT;
	END_VAR
	VAR_INPUT
		(* Indicates the time before the function is cancelled. *)
		nTimeout : TIME := VISION_ADS_TIMEOUT;
	END_VAR
	VAR_OUTPUT
		(* This output remains TRUE until the function block has executed a command, but at the longest for the duration supplied to the 'nTimeout' input. While bBusy = TRUE, no new command will be accepted at the inputs. *)
		bBusy : BOOL;
		(* This output is switched to TRUE as soon as an error occurs during the execution of a command. The command-specific error code is contained in ‘nErrorId’. If the function block has a timeout error, 'bError' is TRUE and 'nErrorId' is 1861 (hexadecimal 0x745). Is reset to FALSE by the execution of a command at the inputs. *)
		bError : BOOL;
	END_VAR
	VAR
		 {attribute 'hide'}
		_reserved2 : UINT;
	END_VAR
	VAR_OUTPUT
		(* Contains the ADS error code or the command-specific error code of the last executed command. Is reset to 0 by the execution of a command at the inputs. *)
		nErrorId : UDINT;
	END_VAR
	VAR
		(* Internal parameter *)
		{attribute 'hide'}
		nAdsInvStamp : UINT;
		(* Internal parameter *)
		{attribute 'hide'}
		nAdsInvCnt : BYTE;
		(* Internal parameter *)
		{attribute 'hide'}
		ePendingRequest : BYTE;
		(* Internal parameter *)
		{attribute 'hide'}
		nTimeElapsed : TIME;
		(* Internal parameter *)
		{attribute 'hide'}
		bLastRead : BOOL;
		 {attribute 'hide'}
		_reserved3 : UINT_24_56;
		(* Internal parameter *)
		{attribute 'hide'}
		 {attribute 'GUID' := '18071995-0000-0000-0000-000000000018'}
		pBuffer : PVOID;
		(* Internal parameter *)
		{attribute 'hide'}
		 {attribute 'GUID' := '18071995-0000-0000-0000-000000000018'}
		pFilePathPending : PVOID;
	END_VAR


	(* Internal method *)
	{attribute 'hide'}
	METHOD FB_exit : BOOL
	VAR_INPUT
		(*  if TRUE, the exit method is called for exiting an instance that is copied afterwards (online change). *)
		bInCopyCode : BOOL;
	END_VAR
END_METHOD


	(* Internal method *)
	{attribute 'hide'}
	METHOD FB_init : BOOL
	VAR_INPUT
		(*  if TRUE, the retain variables are initialized (warm start / cold start) *)
		bInitRetains : BOOL;
		(*  if TRUE, the instance afterwards gets moved into the copy code (online change) *)
		bInCopyCode : BOOL;
	END_VAR
END_METHOD

END_FUNCTION_BLOCK

// Function Blocks/File Access/FB_VN_WriteCalibrationResult

	{attribute 'c++_compatible'}
	{attribute 'external_name' := 'FB_VN_WriteCalibrationResult_GUID_9801AA70_10E4_4F72_CD8B_6EAD6720C926'}
	{attribute 'TcIecLibraryType'}
	(* This FB writes calibration results as a json file to the hard drive. *)
	FUNCTION_BLOCK FB_VN_WriteCalibrationResult
	VAR_IN_OUT CONSTANT
		(* Full path of the file or relative path to the default directory on the target pc (e.g. only a file name). If the string is empty, a file name will be generated (containing the current time). *)
		 {attribute 'GUID' := '18071995-0000-0000-0000-00000000001A'}
		sFilePath : STRING;
	END_VAR
	VAR_INPUT
		(* Returns the camera matrix *)
		 {attribute 'GUID' := '91A420A3-4727-4481-B3BB-170528E5BC7C'}
		 {attribute 'Namespace' := 'VN'}
		aCameraMatrix : REFERENCE TO TcVnMatrix3x3_LREAL;
		(* Returns the distortion coefficients *)
		 {attribute 'GUID' := 'DD112102-C23A-4B37-A43A-A96400B57010'}
		 {attribute 'Namespace' := 'VN'}
		aDistortionCoefficients : REFERENCE TO TcVnArray8_LREAL;
		(* Returns the rotation matrix *)
		 {attribute 'GUID' := '91A420A3-4727-4481-B3BB-170528E5BC7C'}
		 {attribute 'Namespace' := 'VN'}
		aRotationMatrix : REFERENCE TO TcVnMatrix3x3_LREAL;
		(* Returns the translation vector *)
		 {attribute 'GUID' := 'B9A67DEB-A7D1-4F25-95A3-4A82FA5C1E28'}
		 {attribute 'Namespace' := 'VN'}
		aTranslationVector : REFERENCE TO TcVnVector3_LREAL;
		(* Writing the container is triggered by a rising edge at this input. *)
		bWrite : BOOL;
	END_VAR
	VAR
		 {attribute 'hide'}
		_reserved1 : ARRAY [1..3] OF USINT;
	END_VAR
	VAR_INPUT
		(* Indicates the time before the function is cancelled. *)
		nTimeout : TIME := VISION_ADS_TIMEOUT;
	END_VAR
	VAR_OUTPUT
		(* This output remains TRUE until the function block has executed a command, but at the longest for the duration supplied to the 'nTimeout' input. While bBusy = TRUE, no new command will be accepted at the inputs. *)
		bBusy : BOOL;
		(* This output is switched to TRUE as soon as an error occurs during the execution of a command. The command-specific error code is contained in ‘nErrorId’. If the function block has a timeout error, 'bError' is TRUE and 'nErrorId' is 1861 (hexadecimal 0x745). Is reset to FALSE by the execution of a command at the inputs. *)
		bError : BOOL;
	END_VAR
	VAR
		 {attribute 'hide'}
		_reserved2 : UINT;
	END_VAR
	VAR_OUTPUT
		(* Contains the ADS error code or the command-specific error code of the last executed command. Is reset to 0 by the execution of a command at the inputs. *)
		nErrorId : UDINT;
	END_VAR
	VAR
		(* Internal parameter *)
		{attribute 'hide'}
		nAdsInvStamp : UINT;
		(* Internal parameter *)
		{attribute 'hide'}
		nAdsInvCnt : BYTE;
		 {attribute 'hide'}
		_reserved3 : USINT;
		(* Internal parameter *)
		{attribute 'hide'}
		nTimeElapsed : TIME;
		(* Internal parameter *)
		{attribute 'hide'}
		bLastWrite : BOOL;
		 {attribute 'hide'}
		_reserved4 : UINT_24_56;
	END_VAR


	(* Internal method *)
	{attribute 'hide'}
	METHOD FB_exit : BOOL
	VAR_INPUT
		(* If TRUE, the exit method is called for exiting an instance that is copied afterwards (online change). *)
		bInCopyCode : BOOL;
	END_VAR
END_METHOD


	(* Internal method *)
	{attribute 'hide'}
	METHOD FB_init : BOOL
	VAR_INPUT
		(* If TRUE, the retain variables are initialized (warm start / cold start) *)
		bInitRetains : BOOL;
		(* If TRUE, the instance afterwards gets moved into the copy code (online change) *)
		bInCopyCode : BOOL;
	END_VAR
END_METHOD

END_FUNCTION_BLOCK

// Function Blocks/File Access/FB_VN_WriteContainer

	{attribute 'c++_compatible'}
	{attribute 'external_name' := 'FB_VN_WriteContainer_GUID_C9C51CD8_F670_40D9_D8BF_3FDE7F33C30E'}
	{attribute 'TcIecLibraryType'}
	(* This FB writes a container as an xml file to the hard drive. *)
	FUNCTION_BLOCK FB_VN_WriteContainer
	VAR_INPUT
		(* The container to write *)
		 {attribute 'GUID' := 'BC72B333-E095-465B-9693-7979773CA3B8'}
		ipContainer : REFERENCE TO ITcVnContainer;
	END_VAR
	VAR_IN_OUT CONSTANT
		(* Full path of the file or relative path to the default directory on the target pc (e.g. only a file name). If the string is empty, a file name will be generated (containing the current time). *)
		 {attribute 'GUID' := '18071995-0000-0000-0000-00000000001A'}
		sFilePath : STRING;
	END_VAR
	VAR_INPUT
		(* Container export format (default is human readable xml) *)
		 {attribute 'GUID' := 'E9CF1A08-67E7-4F44-A865-987B5AF9C778'}
		 {attribute 'Namespace' := 'Tc3_Vision'}
		eExportFormat : ETcVnContainerExportFormat := TCVN_CEF_XML;
		(* Writing the container is triggered by a rising edge at this input. *)
		bWrite : BOOL;
	END_VAR
	VAR
		 {attribute 'hide'}
		_reserved1 : USINT;
	END_VAR
	VAR_INPUT
		(* Indicates the time before the function is cancelled. *)
		nTimeout : TIME := VISION_ADS_TIMEOUT;
	END_VAR
	VAR_OUTPUT
		(* This output remains TRUE until the function block has executed a command, but at the longest for the duration supplied to the 'nTimeout' input. While bBusy = TRUE, no new command will be accepted at the inputs. *)
		bBusy : BOOL;
		(* This output is switched to TRUE as soon as an error occurs during the execution of a command. The command-specific error code is contained in ‘nErrorId’. If the function block has a timeout error, 'bError' is TRUE and 'nErrorId' is 1861 (hexadecimal 0x745). Is reset to FALSE by the execution of a command at the inputs. *)
		bError : BOOL;
	END_VAR
	VAR
		 {attribute 'hide'}
		_reserved2 : UINT;
	END_VAR
	VAR_OUTPUT
		(* Contains the ADS error code or the command-specific error code of the last executed command. Is reset to 0 by the execution of a command at the inputs. *)
		nErrorId : UDINT;
	END_VAR
	VAR
		(* Internal parameter *)
		{attribute 'hide'}
		nAdsInvStamp : UINT;
		(* Internal parameter *)
		{attribute 'hide'}
		nAdsInvCnt : BYTE;
		 {attribute 'hide'}
		_reserved3 : USINT;
		(* Internal parameter *)
		{attribute 'hide'}
		nTimeElapsed : TIME;
		(* Internal parameter *)
		{attribute 'hide'}
		bLastWrite : BOOL;
		 {attribute 'hide'}
		_reserved4 : UINT_24_56;
	END_VAR


	(* Internal method *)
	{attribute 'hide'}
	METHOD FB_exit : BOOL
	VAR_INPUT
		(* If TRUE, the exit method is called for exiting an instance that is copied afterwards (online change). *)
		bInCopyCode : BOOL;
	END_VAR
END_METHOD


	(* Internal method *)
	{attribute 'hide'}
	METHOD FB_init : BOOL
	VAR_INPUT
		(* If TRUE, the retain variables are initialized (warm start / cold start) *)
		bInitRetains : BOOL;
		(* If TRUE, the instance afterwards gets moved into the copy code (online change) *)
		bInCopyCode : BOOL;
	END_VAR
END_METHOD

END_FUNCTION_BLOCK

// Function Blocks/File Access/FB_VN_WriteImage

	{attribute 'c++_compatible'}
	{attribute 'external_name' := 'FB_VN_WriteImage_GUID_27C557F6_6D7B_4C1E_D96C_8B0E5D26785B'}
	{attribute 'TcIecLibraryType'}
	(* This FB writes an image to the hard drive. *)
	FUNCTION_BLOCK FB_VN_WriteImage
	VAR_INPUT
		(* The image to write *)
		 {attribute 'GUID' := '70D42C6D-6F4E-4719-8B29-2883D5D59B1C'}
		ipImage : REFERENCE TO ITcVnImage;
	END_VAR
	VAR_IN_OUT CONSTANT
		(* Full path of the file or relative path to the default directory on the target pc (e.g. only a file name). If the string is empty, a file name will be generated (containing the current time). *)
		 {attribute 'GUID' := '18071995-0000-0000-0000-00000000001A'}
		sFilePath : STRING;
	END_VAR
	VAR_INPUT
		(* Writing the image is triggered by a rising edge at this input. *)
		bWrite : BOOL;
	END_VAR
	VAR
		 {attribute 'hide'}
		_reserved1 : ARRAY [1..3] OF USINT;
	END_VAR
	VAR_INPUT
		(* Indicates the time before the function is cancelled. *)
		nTimeout : TIME := VISION_ADS_TIMEOUT;
	END_VAR
	VAR_OUTPUT
		(* This output remains TRUE until the function block has executed a command, but at the longest for the duration supplied to the 'nTimeout' input. While bBusy = TRUE, no new command will be accepted at the inputs. *)
		bBusy : BOOL;
		(* This output is switched to TRUE as soon as an error occurs during the execution of a command. The command-specific error code is contained in ‘nErrorId’. If the function block has a timeout error, 'bError' is TRUE and 'nErrorId' is 1861 (hexadecimal 0x745). Is reset to FALSE by the execution of a command at the inputs. *)
		bError : BOOL;
	END_VAR
	VAR
		 {attribute 'hide'}
		_reserved2 : UINT;
	END_VAR
	VAR_OUTPUT
		(* Contains the ADS error code or the command-specific error code of the last executed command. Is reset to 0 by the execution of a command at the inputs. *)
		nErrorId : UDINT;
	END_VAR
	VAR
		(* Internal parameter *)
		{attribute 'hide'}
		nAdsInvStamp : UINT;
		(* Internal parameter *)
		{attribute 'hide'}
		nAdsInvCnt : BYTE;
		 {attribute 'hide'}
		_reserved3 : USINT;
		(* Internal parameter *)
		{attribute 'hide'}
		nTimeElapsed : TIME;
		(* Internal parameter *)
		{attribute 'hide'}
		bLastWrite : BOOL;
		 {attribute 'hide'}
		_reserved4 : UINT_24_56;
	END_VAR


	(* Internal method *)
	{attribute 'hide'}
	METHOD FB_exit : BOOL
	VAR_INPUT
		(*  if TRUE, the exit method is called for exiting an instance that is copied afterwards (online change). *)
		bInCopyCode : BOOL;
	END_VAR
END_METHOD


	(* Internal method *)
	{attribute 'hide'}
	METHOD FB_init : BOOL
	VAR_INPUT
		(*  if TRUE, the retain variables are initialized (warm start / cold start) *)
		bInitRetains : BOOL;
		(*  if TRUE, the instance afterwards gets moved into the copy code (online change) *)
		bInCopyCode : BOOL;
	END_VAR
END_METHOD

END_FUNCTION_BLOCK

// Function Blocks/File Access/FB_VN_WriteMlModel

	{attribute 'c++_compatible'}
	{attribute 'external_name' := 'FB_VN_WriteMlModel_GUID_A98A6DC4_C377_45E6_FC7D_68B89096C74C'}
	{attribute 'TcIecLibraryType'}
	(* This FB writes a machine learning model to the hard drive. *)
	FUNCTION_BLOCK FB_VN_WriteMlModel
	VAR_INPUT
		(* The machine learning model to write *)
		 {attribute 'GUID' := 'AC23D64B-CDFA-4D43-AE8B-364A856EB3E2'}
		ipMlModel : REFERENCE TO ITcVnMlModel;
	END_VAR
	VAR_IN_OUT CONSTANT
		(* Full path of the file or relative path to the default directory on the target pc (e.g. only a file name). If the string is empty, a file name will be generated (containing the current time). *)
		 {attribute 'GUID' := '18071995-0000-0000-0000-00000000001A'}
		sFilePath : STRING;
	END_VAR
	VAR_INPUT
		(* Writing the machine learning model is triggered by a rising edge at this input. *)
		bWrite : BOOL;
	END_VAR
	VAR
		 {attribute 'hide'}
		_reserved1 : ARRAY [1..3] OF USINT;
	END_VAR
	VAR_INPUT
		(* Indicates the time before the function is cancelled. *)
		nTimeout : TIME := VISION_ADS_TIMEOUT;
	END_VAR
	VAR_OUTPUT
		(* This output remains TRUE until the function block has executed a command, but at the longest for the duration supplied to the 'nTimeout' input. While bBusy = TRUE, no new command will be accepted at the inputs. *)
		bBusy : BOOL;
		(* This output is switched to TRUE as soon as an error occurs during the execution of a command. The command-specific error code is contained in ‘nErrorId’. If the function block has a timeout error, 'bError' is TRUE and 'nErrorId' is 1861 (hexadecimal 0x745). Is reset to FALSE by the execution of a command at the inputs. *)
		bError : BOOL;
	END_VAR
	VAR
		 {attribute 'hide'}
		_reserved2 : UINT;
	END_VAR
	VAR_OUTPUT
		(* Contains the ADS error code or the command-specific error code of the last executed command. Is reset to 0 by the execution of a command at the inputs. *)
		nErrorId : UDINT;
	END_VAR
	VAR
		(* Internal parameter *)
		{attribute 'hide'}
		nAdsInvStamp : UINT;
		(* Internal parameter *)
		{attribute 'hide'}
		nAdsInvCnt : BYTE;
		 {attribute 'hide'}
		_reserved3 : USINT;
		(* Internal parameter *)
		{attribute 'hide'}
		nTimeElapsed : TIME;
		(* Internal parameter *)
		{attribute 'hide'}
		bLastWrite : BOOL;
		 {attribute 'hide'}
		_reserved4 : UINT_24_56;
	END_VAR


	(* Internal method *)
	{attribute 'hide'}
	METHOD FB_exit : BOOL
	VAR_INPUT
		(*  if TRUE, the exit method is called for exiting an instance that is copied afterwards (online change). *)
		bInCopyCode : BOOL;
	END_VAR
END_METHOD


	(* Internal method *)
	{attribute 'hide'}
	METHOD FB_init : BOOL
	VAR_INPUT
		(*  if TRUE, the retain variables are initialized (warm start / cold start) *)
		bInitRetains : BOOL;
		(*  if TRUE, the instance afterwards gets moved into the copy code (online change) *)
		bInCopyCode : BOOL;
	END_VAR
END_METHOD

END_FUNCTION_BLOCK

// Function Blocks/Camera Register Access/FB_VN_ReadRegister_UDINT

	{attribute 'c++_compatible'}
	{attribute 'external_name' := 'FB_VN_ReadRegister_UDINT_GUID_36306262_B8AC_4335_C4EC_00A9B7592AFE'}
	{attribute 'TcIecLibraryType'}
	(* This FB reads a DINT register from the camera. Requires an open control channel (e.g. by calling FB_VN_GevCameraControl.OpenCamera() before) *)
	FUNCTION_BLOCK FB_VN_ReadRegister_UDINT
	VAR_INPUT
		(* The address of the register that should be read *)
		 {attribute 'GUID' := 'E1ED2436-3512-43FA-B927-3F71DEDDA853'}
		nAddress : GVCP_REGISTER_ADDRESS;
		(* OPTIONAL: The endianness of the register. 0 = Big, 1 = Little. Default: 0 *)
		nEndian : UINT;
		(* Reading the register is triggered by a rising edge at this input. *)
		bRead : BOOL;
	END_VAR
	VAR
		 {attribute 'hide'}
		_reserved1 : USINT;
	END_VAR
	VAR_INPUT
		(* Indicates the time before the function is cancelled. *)
		nTimeout : TIME := VISION_ADS_TIMEOUT;
	END_VAR
	VAR_OUTPUT
		(* The read value *)
		nValue : UDINT;
		(* This output remains TRUE until the function block has executed a command, but at the longest for the duration supplied to the 'nTimeout' input. While bBusy = TRUE, no new command will be accepted at the inputs. *)
		bBusy : BOOL;
		(* This output is switched to TRUE as soon as an error occurs during the execution of a command. The command-specific error code is contained in ‘nErrorId’. If the function block has a timeout error, 'bError' is TRUE and 'nErrorId' is 1861 (hexadecimal 0x745). Is reset to FALSE by the execution of a command at the inputs. *)
		bError : BOOL;
	END_VAR
	VAR
		 {attribute 'hide'}
		_reserved2 : UINT;
	END_VAR
	VAR_OUTPUT
		(* Contains the ADS error code or the command-specific error code of the last executed command. Is reset to 0 by the execution of a command at the inputs. *)
		nErrorId : UDINT;
	END_VAR
	VAR
		(* Internal reference to the corresponding TcVnGevImageProvider TcCOM module ID, which needs to be set via TC init symbol. *)
		{attribute 'TcInitSymbol'}
		{attribute 'TcCategoryOID' := 'TcVnGevImageProvider'}
		 {attribute 'GUID' := '18071995-0000-0000-0000-00000000000F'}
		oidITcVnGevImageProvider : OTCID;
		 {attribute 'hide'}
		_reserved3 : UINT_0_32;
		(* Internal reference to the corresponding TcVnGevImageProvider module. *)
		{attribute 'hide'}
		 {attribute 'GUID' := 'ED7659DB-95DC-4A4A-B62F-02C9870D5E81'}
		ipGevImageProvider : ITcVnGevImageProvider;
		(* Internal timestamp for timeout detection *)
		{attribute 'hide'}
		nTimeElapsed : TIME;
		(* Internal flag for rising edge detection *)
		{attribute 'hide'}
		bLastRead : BOOL;
		 {attribute 'hide'}
		_reserved4 : ARRAY [1..3] OF USINT;
	END_VAR


	(* Internal method *)
	{attribute 'hide'}
	METHOD FB_exit : BOOL
	VAR_INPUT
		(*  if TRUE, the exit method is called for exiting an instance that is copied afterwards (online change). *)
		bInCopyCode : BOOL;
	END_VAR
END_METHOD


	(* Internal method *)
	{attribute 'hide'}
	METHOD FB_init : BOOL
	VAR_INPUT
		(*  if TRUE, the retain variables are initialized (warm start / cold start) *)
		bInitRetains : BOOL;
		(*  if TRUE, the instance afterwards gets moved into the copy code (online change) *)
		bInCopyCode : BOOL;
	END_VAR
END_METHOD

END_FUNCTION_BLOCK

// Function Blocks/Camera Register Access/FB_VN_WriteRegister_UDINT

	{attribute 'c++_compatible'}
	{attribute 'external_name' := 'FB_VN_WriteRegister_UDINT_GUID_286C50FA_63EF_4997_DA2E_6E63159DC45C'}
	{attribute 'TcIecLibraryType'}
	(* This FB writes a DINT value into a register on the camera. Requires an open control channel (e.g. by calling FB_VN_GevCameraControl.OpenCamera() before) *)
	FUNCTION_BLOCK FB_VN_WriteRegister_UDINT
	VAR_INPUT
		(* The address of the register that should be written *)
		 {attribute 'GUID' := 'E1ED2436-3512-43FA-B927-3F71DEDDA853'}
		nAddress : GVCP_REGISTER_ADDRESS;
		(* The value to write *)
		nValue : UDINT;
		(* OPTIONAL: The endianness of the register. 0 = Big, 1 = Little. Default: 0 *)
		nEndian : UINT;
		(* Writing the register is triggered by a rising edge at this input. *)
		bWrite : BOOL;
	END_VAR
	VAR
		 {attribute 'hide'}
		_reserved1 : USINT;
	END_VAR
	VAR_INPUT
		(* Indicates the time before the function is cancelled. *)
		nTimeout : TIME := VISION_ADS_TIMEOUT;
	END_VAR
	VAR_OUTPUT
		(* This output remains TRUE until the function block has executed a command, but at the longest for the duration supplied to the 'nTimeout' input. While bBusy = TRUE, no new command will be accepted at the inputs. *)
		bBusy : BOOL;
		(* This output is switched to TRUE as soon as an error occurs during the execution of a command. The command-specific error code is contained in ‘nErrorId’. If the function block has a timeout error, 'bError' is TRUE and 'nErrorId' is 1861 (hexadecimal 0x745). Is reset to FALSE by the execution of a command at the inputs. *)
		bError : BOOL;
	END_VAR
	VAR
		 {attribute 'hide'}
		_reserved2 : UINT;
	END_VAR
	VAR_OUTPUT
		(* Contains the ADS error code or the command-specific error code of the last executed command. Is reset to 0 by the execution of a command at the inputs. *)
		nErrorId : UDINT;
	END_VAR
	VAR
		(* Internal reference to the corresponding TcVnGevImageProvider TcCOM module ID, which needs to be set via TC init symbol. *)
		{attribute 'TcInitSymbol'}
		{attribute 'TcCategoryOID' := 'TcVnGevImageProvider'}
		 {attribute 'GUID' := '18071995-0000-0000-0000-00000000000F'}
		oidITcVnGevImageProvider : OTCID;
		 {attribute 'hide'}
		_reserved3 : UINT_0_32;
		(* Internal reference to the corresponding TcVnGevImageProvider module. *)
		{attribute 'hide'}
		 {attribute 'GUID' := 'ED7659DB-95DC-4A4A-B62F-02C9870D5E81'}
		ipGevImageProvider : ITcVnGevImageProvider;
		(* Internal timestamp for timeout detection *)
		{attribute 'hide'}
		nTimeElapsed : TIME;
		(* Internal flag for rising edge detection *)
		{attribute 'hide'}
		bLastWrite : BOOL;
		 {attribute 'hide'}
		_reserved4 : ARRAY [1..3] OF USINT;
	END_VAR


	(* Internal method *)
	{attribute 'hide'}
	METHOD FB_exit : BOOL
	VAR_INPUT
		(*  if TRUE, the exit method is called for exiting an instance that is copied afterwards (online change). *)
		bInCopyCode : BOOL;
	END_VAR
END_METHOD


	(* Internal method *)
	{attribute 'hide'}
	METHOD FB_init : BOOL
	VAR_INPUT
		(*  if TRUE, the retain variables are initialized (warm start / cold start) *)
		bInitRetains : BOOL;
		(*  if TRUE, the instance afterwards gets moved into the copy code (online change) *)
		bInCopyCode : BOOL;
	END_VAR
END_METHOD

END_FUNCTION_BLOCK

// Function Blocks/Camera Register Access/FB_VN_ReadRegister_ULINT

	{attribute 'c++_compatible'}
	{attribute 'external_name' := 'FB_VN_ReadRegister_ULINT_GUID_EA62D868_8248_4DDD_CF69_EA64F98B531B'}
	{attribute 'TcIecLibraryType'}
	(* This FB reads a ULINT register from the camera. Requires an open control channel (e.g. by calling FB_VN_GevCameraControl.OpenCamera() before) *)
	FUNCTION_BLOCK FB_VN_ReadRegister_ULINT
	VAR_INPUT
		(* The address of the register that should be read *)
		 {attribute 'GUID' := 'E1ED2436-3512-43FA-B927-3F71DEDDA853'}
		nAddress : GVCP_REGISTER_ADDRESS;
		(* OPTIONAL: The endianness of the register. 0 = Big, 1 = Little. Default: 0 *)
		nEndian : UINT;
		(* Reading the register is triggered by a rising edge at this input. *)
		bRead : BOOL;
	END_VAR
	VAR
		 {attribute 'hide'}
		_reserved1 : USINT;
	END_VAR
	VAR_INPUT
		(* Indicates the time before the function is cancelled. *)
		nTimeout : TIME := VISION_ADS_TIMEOUT;
	END_VAR
	VAR
		 {attribute 'hide'}
		_reserved2 : UINT_0_32;
	END_VAR
	VAR_OUTPUT
		(* The read value *)
		nValue : ULINT;
		(* This output remains TRUE until the function block has executed a command, but at the longest for the duration supplied to the 'nTimeout' input. While bBusy = TRUE, no new command will be accepted at the inputs. *)
		bBusy : BOOL;
		(* This output is switched to TRUE as soon as an error occurs during the execution of a command. The command-specific error code is contained in ‘nErrorId’. If the function block has a timeout error, 'bError' is TRUE and 'nErrorId' is 1861 (hexadecimal 0x745). Is reset to FALSE by the execution of a command at the inputs. *)
		bError : BOOL;
	END_VAR
	VAR
		 {attribute 'hide'}
		_reserved3 : UINT;
	END_VAR
	VAR_OUTPUT
		(* Contains the ADS error code or the command-specific error code of the last executed command. Is reset to 0 by the execution of a command at the inputs. *)
		nErrorId : UDINT;
	END_VAR
	VAR
		(* Internal reference to the corresponding TcVnGevImageProvider TcCOM module ID, which needs to be set via TC init symbol. *)
		{attribute 'TcInitSymbol'}
		{attribute 'TcCategoryOID' := 'TcVnGevImageProvider'}
		 {attribute 'GUID' := '18071995-0000-0000-0000-00000000000F'}
		oidITcVnGevImageProvider : OTCID;
		 {attribute 'hide'}
		_reserved4 : UINT_0_32;
		(* Internal reference to the corresponding TcVnGevImageProvider module. *)
		{attribute 'hide'}
		 {attribute 'GUID' := 'ED7659DB-95DC-4A4A-B62F-02C9870D5E81'}
		ipGevImageProvider : ITcVnGevImageProvider;
		(* Internal timestamp for timeout detection *)
		{attribute 'hide'}
		nTimeElapsed : TIME;
		(* Internal flag for rising edge detection *)
		{attribute 'hide'}
		bLastRead : BOOL;
		 {attribute 'hide'}
		_reserved5 : ARRAY [1..3] OF USINT;
	END_VAR


	(* Internal method *)
	{attribute 'hide'}
	METHOD FB_exit : BOOL
	VAR_INPUT
		(*  if TRUE, the exit method is called for exiting an instance that is copied afterwards (online change). *)
		bInCopyCode : BOOL;
	END_VAR
END_METHOD


	(* Internal method *)
	{attribute 'hide'}
	METHOD FB_init : BOOL
	VAR_INPUT
		(*  if TRUE, the retain variables are initialized (warm start / cold start) *)
		bInitRetains : BOOL;
		(*  if TRUE, the instance afterwards gets moved into the copy code (online change) *)
		bInCopyCode : BOOL;
	END_VAR
END_METHOD

END_FUNCTION_BLOCK

// Function Blocks/Camera Register Access/FB_VN_WriteRegister_ULINT

	{attribute 'c++_compatible'}
	{attribute 'external_name' := 'FB_VN_WriteRegister_ULINT_GUID_7234D37E_43B2_41CE_E645_9A55A2187C2D'}
	{attribute 'TcIecLibraryType'}
	(* This FB writes a ULINT value into a register on the camera. Requires an open control channel (e.g. by calling FB_VN_GevCameraControl.OpenCamera() before) *)
	FUNCTION_BLOCK FB_VN_WriteRegister_ULINT
	VAR_INPUT
		(* The address of the register that should be written *)
		 {attribute 'GUID' := 'E1ED2436-3512-43FA-B927-3F71DEDDA853'}
		nAddress : GVCP_REGISTER_ADDRESS;
	END_VAR
	VAR
		 {attribute 'hide'}
		_reserved1 : UINT_0_32;
	END_VAR
	VAR_INPUT
		(* The value to write *)
		nValue : ULINT;
		(* OPTIONAL: The endianness of the register. 0 = Big, 1 = Little. Default: 0 *)
		nEndian : UINT;
		(* Writing the register is triggered by a rising edge at this input. *)
		bWrite : BOOL;
	END_VAR
	VAR
		 {attribute 'hide'}
		_reserved2 : USINT;
	END_VAR
	VAR_INPUT
		(* Indicates the time before the function is cancelled. *)
		nTimeout : TIME := VISION_ADS_TIMEOUT;
	END_VAR
	VAR_OUTPUT
		(* This output remains TRUE until the function block has executed a command, but at the longest for the duration supplied to the 'nTimeout' input. While bBusy = TRUE, no new command will be accepted at the inputs. *)
		bBusy : BOOL;
		(* This output is switched to TRUE as soon as an error occurs during the execution of a command. The command-specific error code is contained in ‘nErrorId’. If the function block has a timeout error, 'bError' is TRUE and 'nErrorId' is 1861 (hexadecimal 0x745). Is reset to FALSE by the execution of a command at the inputs. *)
		bError : BOOL;
	END_VAR
	VAR
		 {attribute 'hide'}
		_reserved3 : UINT;
	END_VAR
	VAR_OUTPUT
		(* Contains the ADS error code or the command-specific error code of the last executed command. Is reset to 0 by the execution of a command at the inputs. *)
		nErrorId : UDINT;
	END_VAR
	VAR
		(* Internal reference to the corresponding TcVnGevImageProvider TcCOM module ID, which needs to be set via TC init symbol. *)
		{attribute 'TcInitSymbol'}
		{attribute 'TcCategoryOID' := 'TcVnGevImageProvider'}
		 {attribute 'GUID' := '18071995-0000-0000-0000-00000000000F'}
		oidITcVnGevImageProvider : OTCID;
		 {attribute 'hide'}
		_reserved4 : UINT_0_32;
		(* Internal reference to the corresponding TcVnGevImageProvider module. *)
		{attribute 'hide'}
		 {attribute 'GUID' := 'ED7659DB-95DC-4A4A-B62F-02C9870D5E81'}
		ipGevImageProvider : ITcVnGevImageProvider;
		(* Internal timestamp for timeout detection *)
		{attribute 'hide'}
		nTimeElapsed : TIME;
		(* Internal flag for rising edge detection *)
		{attribute 'hide'}
		bLastWrite : BOOL;
		 {attribute 'hide'}
		_reserved5 : ARRAY [1..3] OF USINT;
	END_VAR


	(* Internal method *)
	{attribute 'hide'}
	METHOD FB_exit : BOOL
	VAR_INPUT
		(*  if TRUE, the exit method is called for exiting an instance that is copied afterwards (online change). *)
		bInCopyCode : BOOL;
	END_VAR
END_METHOD


	(* Internal method *)
	{attribute 'hide'}
	METHOD FB_init : BOOL
	VAR_INPUT
		(*  if TRUE, the retain variables are initialized (warm start / cold start) *)
		bInitRetains : BOOL;
		(*  if TRUE, the instance afterwards gets moved into the copy code (online change) *)
		bInCopyCode : BOOL;
	END_VAR
END_METHOD

END_FUNCTION_BLOCK

// Function Blocks/Camera Register Access/FB_VN_ReadMemory

